        recipe definition RecGroup: arScrew[0].rRstmax : REAL; arScrew[0].rRstmin : REAL; arScrew[0].iCountCycle : INT; arScrew[0].iActuatorsMove : INT; arScrew[0].iActuatorsStep : INT; arScrew[0].iActuatorsStartPos[0] : INT; arScrew[0].iActuatorsStartPos[1] : INT; arScrew[0].support[0].bPosition : BOOL; arScrew[0].support[0].arLength[0] : INT; arScrew[0].support[0].arLength[1] : INT; arScrew[0].support[0].name : WSTRING(20); arScrew[0].support[1].bPosition : BOOL; arScrew[0].support[1].arLength[0] : INT; arScrew[0].support[1].arLength[1] : INT; arScrew[0].support[1].name : WSTRING(20); arScrew[0].bDirRotate : BOOL; arScrew[0].rOut_diam : REAL; arScrew[0].rInner_diam : REAL; arScrew[0].rTurn_step : REAL; arScrew[0].rWidth : REAL; arScrew[0].rAngle_knives : REAL; arScrew[0].rMidle_line : REAL; arScrew[0].rInstal_support : REAL; arScrew[0].rPosX0 : REAL; arScrew[0].rPosX1 : REAL; arScrew[0].rPosX2 : REAL; arScrew[0].equip.place : WSTRING(10); arScrew[0].equip.name : WSTRING(20); arScrew[0].name : WSTRING(20); arScrew[1].rRstmax : REAL; arScrew[1].rRstmin : REAL; arScrew[1].iCountCycle : INT; arScrew[1].iActuatorsMove : INT; arScrew[1].iActuatorsStep : INT; arScrew[1].iActuatorsStartPos[0] : INT; arScrew[1].iActuatorsStartPos[1] : INT; arScrew[1].support[0].bPosition : BOOL; arScrew[1].support[0].arLength[0] : INT; arScrew[1].support[0].arLength[1] : INT; arScrew[1].support[0].name : WSTRING(20); arScrew[1].support[1].bPosition : BOOL; arScrew[1].support[1].arLength[0] : INT; arScrew[1].support[1].arLength[1] : INT; arScrew[1].support[1].name : WSTRING(20); arScrew[1].bDirRotate : BOOL; arScrew[1].rOut_diam : REAL; arScrew[1].rInner_diam : REAL; arScrew[1].rTurn_step : REAL; arScrew[1].rWidth : REAL; arScrew[1].rAngle_knives : REAL; arScrew[1].rMidle_line : REAL; arScrew[1].rInstal_support : REAL; arScrew[1].rPosX0 : REAL; arScrew[1].rPosX1 : REAL; arScrew[1].rPosX2 : REAL; arScrew[1].equip.place : WSTRING(10); arScrew[1].equip.name : WSTRING(20); arScrew[1].name : WSTRING(20); arScrew[2].rRstmax : REAL; arScrew[2].rRstmin : REAL; arScrew[2].iCountCycle : INT; arScrew[2].iActuatorsMove : INT; arScrew[2].iActuatorsStep : INT; arScrew[2].iActuatorsStartPos[0] : INT; arScrew[2].iActuatorsStartPos[1] : INT; arScrew[2].support[0].bPosition : BOOL; arScrew[2].support[0].arLength[0] : INT; arScrew[2].support[0].arLength[1] : INT; arScrew[2].support[0].name : WSTRING(20); arScrew[2].support[1].bPosition : BOOL; arScrew[2].support[1].arLength[0] : INT; arScrew[2].support[1].arLength[1] : INT; arScrew[2].support[1].name : WSTRING(20); arScrew[2].bDirRotate : BOOL; arScrew[2].rOut_diam : REAL; arScrew[2].rInner_diam : REAL; arScrew[2].rTurn_step : REAL; arScrew[2].rWidth : REAL; arScrew[2].rAngle_knives : REAL; arScrew[2].rMidle_line : REAL; arScrew[2].rInstal_support : REAL; arScrew[2].rPosX0 : REAL; arScrew[2].rPosX1 : REAL; arScrew[2].rPosX2 : REAL; arScrew[2].equip.place : WSTRING(10); arScrew[2].equip.name : WSTRING(20); arScrew[2].name : WSTRING(20); arScrew[3].rRstmax : REAL; arScrew[3].rRstmin : REAL; arScrew[3].iCountCycle : INT; arScrew[3].iActuatorsMove : INT; arScrew[3].iActuatorsStep : INT; arScrew[3].iActuatorsStartPos[0] : INT; arScrew[3].iActuatorsStartPos[1] : INT; arScrew[3].support[0].bPosition : BOOL; arScrew[3].support[0].arLength[0] : INT; arScrew[3].support[0].arLength[1] : INT; arScrew[3].support[0].name : WSTRING(20); arScrew[3].support[1].bPosition : BOOL; arScrew[3].support[1].arLength[0] : INT; arScrew[3].support[1].arLength[1] : INT; arScrew[3].support[1].name : WSTRING(20); arScrew[3].bDirRotate : BOOL; arScrew[3].rOut_diam : REAL; arScrew[3].rInner_diam : REAL; arScrew[3].rTurn_step : REAL; arScrew[3].rWidth : REAL; arScrew[3].rAngle_knives : REAL; arScrew[3].rMidle_line : REAL; arScrew[3].rInstal_support : REAL; arScrew[3].rPosX0 : REAL; arScrew[3].rPosX1 : REAL; arScrew[3].rPosX2 : REAL; arScrew[3].equip.place : WSTRING(10); arScrew[3].equip.name : WSTRING(20); arScrew[3].name : WSTRING(20); arScrew[4].rRstmax : REAL; arScrew[4].rRstmin : REAL; arScrew[4].iCountCycle : INT; arScrew[4].iActuatorsMove : INT; arScrew[4].iActuatorsStep : INT; arScrew[4].iActuatorsStartPos[0] : INT; arScrew[4].iActuatorsStartPos[1] : INT; arScrew[4].support[0].bPosition : BOOL; arScrew[4].support[0].arLength[0] : INT; arScrew[4].support[0].arLength[1] : INT; arScrew[4].support[0].name : WSTRING(20); arScrew[4].support[1].bPosition : BOOL; arScrew[4].support[1].arLength[0] : INT; arScrew[4].support[1].arLength[1] : INT; arScrew[4].support[1].name : WSTRING(20); arScrew[4].bDirRotate : BOOL; arScrew[4].rOut_diam : REAL; arScrew[4].rInner_diam : REAL; arScrew[4].rTurn_step : REAL; arScrew[4].rWidth : REAL; arScrew[4].rAngle_knives : REAL; arScrew[4].rMidle_line : REAL; arScrew[4].rInstal_support : REAL; arScrew[4].rPosX0 : REAL; arScrew[4].rPosX1 : REAL; arScrew[4].rPosX2 : REAL; arScrew[4].equip.place : WSTRING(10); arScrew[4].equip.name : WSTRING(20); arScrew[4].name : WSTRING(20); arScrew[5].rRstmax : REAL; arScrew[5].rRstmin : REAL; arScrew[5].iCountCycle : INT; arScrew[5].iActuatorsMove : INT; arScrew[5].iActuatorsStep : INT; arScrew[5].iActuatorsStartPos[0] : INT; arScrew[5].iActuatorsStartPos[1] : INT; arScrew[5].support[0].bPosition : BOOL; arScrew[5].support[0].arLength[0] : INT; arScrew[5].support[0].arLength[1] : INT; arScrew[5].support[0].name : WSTRING(20); arScrew[5].support[1].bPosition : BOOL; arScrew[5].support[1].arLength[0] : INT; arScrew[5].support[1].arLength[1] : INT; arScrew[5].support[1].name : WSTRING(20); arScrew[5].bDirRotate : BOOL; arScrew[5].rOut_diam : REAL; arScrew[5].rInner_diam : REAL; arScrew[5].rTurn_step : REAL; arScrew[5].rWidth : REAL; arScrew[5].rAngle_knives : REAL; arScrew[5].rMidle_line : REAL; arScrew[5].rInstal_support : REAL; arScrew[5].rPosX0 : REAL; arScrew[5].rPosX1 : REAL; arScrew[5].rPosX2 : REAL; arScrew[5].equip.place : WSTRING(10); arScrew[5].equip.name : WSTRING(20); arScrew[5].name : WSTRING(20); arScrew[6].rRstmax : REAL; arScrew[6].rRstmin : REAL; arScrew[6].iCountCycle : INT; arScrew[6].iActuatorsMove : INT; arScrew[6].iActuatorsStep : INT; arScrew[6].iActuatorsStartPos[0] : INT; arScrew[6].iActuatorsStartPos[1] : INT; arScrew[6].support[0].bPosition : BOOL; arScrew[6].support[0].arLength[0] : INT; arScrew[6].support[0].arLength[1] : INT; arScrew[6].support[0].name : WSTRING(20); arScrew[6].support[1].bPosition : BOOL; arScrew[6].support[1].arLength[0] : INT; arScrew[6].support[1].arLength[1] : INT; arScrew[6].support[1].name : WSTRING(20); arScrew[6].bDirRotate : BOOL; arScrew[6].rOut_diam : REAL; arScrew[6].rInner_diam : REAL; arScrew[6].rTurn_step : REAL; arScrew[6].rWidth : REAL; arScrew[6].rAngle_knives : REAL; arScrew[6].rMidle_line : REAL; arScrew[6].rInstal_support : REAL; arScrew[6].rPosX0 : REAL; arScrew[6].rPosX1 : REAL; arScrew[6].rPosX2 : REAL; arScrew[6].equip.place : WSTRING(10); arScrew[6].equip.name : WSTRING(20); arScrew[6].name : WSTRING(20); arScrew[7].rRstmax : REAL; arScrew[7].rRstmin : REAL; arScrew[7].iCountCycle : INT; arScrew[7].iActuatorsMove : INT; arScrew[7].iActuatorsStep : INT; arScrew[7].iActuatorsStartPos[0] : INT; arScrew[7].iActuatorsStartPos[1] : INT; arScrew[7].support[0].bPosition : BOOL; arScrew[7].support[0].arLength[0] : INT; arScrew[7].support[0].arLength[1] : INT; arScrew[7].support[0].name : WSTRING(20); arScrew[7].support[1].bPosition : BOOL; arScrew[7].support[1].arLength[0] : INT; arScrew[7].support[1].arLength[1] : INT; arScrew[7].support[1].name : WSTRING(20); arScrew[7].bDirRotate : BOOL; arScrew[7].rOut_diam : REAL; arScrew[7].rInner_diam : REAL; arScrew[7].rTurn_step : REAL; arScrew[7].rWidth : REAL; arScrew[7].rAngle_knives : REAL; arScrew[7].rMidle_line : REAL; arScrew[7].rInstal_support : REAL; arScrew[7].rPosX0 : REAL; arScrew[7].rPosX1 : REAL; arScrew[7].rPosX2 : REAL; arScrew[7].equip.place : WSTRING(10); arScrew[7].equip.name : WSTRING(20); arScrew[7].name : WSTRING(20); arScrew[8].rRstmax : REAL; arScrew[8].rRstmin : REAL; arScrew[8].iCountCycle : INT; arScrew[8].iActuatorsMove : INT; arScrew[8].iActuatorsStep : INT; arScrew[8].iActuatorsStartPos[0] : INT; arScrew[8].iActuatorsStartPos[1] : INT; arScrew[8].support[0].bPosition : BOOL; arScrew[8].support[0].arLength[0] : INT; arScrew[8].support[0].arLength[1] : INT; arScrew[8].support[0].name : WSTRING(20); arScrew[8].support[1].bPosition : BOOL; arScrew[8].support[1].arLength[0] : INT; arScrew[8].support[1].arLength[1] : INT; arScrew[8].support[1].name : WSTRING(20); arScrew[8].bDirRotate : BOOL; arScrew[8].rOut_diam : REAL; arScrew[8].rInner_diam : REAL; arScrew[8].rTurn_step : REAL; arScrew[8].rWidth : REAL; arScrew[8].rAngle_knives : REAL; arScrew[8].rMidle_line : REAL; arScrew[8].rInstal_support : REAL; arScrew[8].rPosX0 : REAL; arScrew[8].rPosX1 : REAL; arScrew[8].rPosX2 : REAL; arScrew[8].equip.place : WSTRING(10); arScrew[8].equip.name : WSTRING(20); arScrew[8].name : WSTRING(20); arScrew[9].rRstmax : REAL; arScrew[9].rRstmin : REAL; arScrew[9].iCountCycle : INT; arScrew[9].iActuatorsMove : INT; arScrew[9].iActuatorsStep : INT; arScrew[9].iActuatorsStartPos[0] : INT; arScrew[9].iActuatorsStartPos[1] : INT; arScrew[9].support[0].bPosition : BOOL; arScrew[9].support[0].arLength[0] : INT; arScrew[9].support[0].arLength[1] : INT; arScrew[9].support[0].name : WSTRING(20); arScrew[9].support[1].bPosition : BOOL; arScrew[9].support[1].arLength[0] : INT; arScrew[9].support[1].arLength[1] : INT; arScrew[9].support[1].name : WSTRING(20); arScrew[9].bDirRotate : BOOL; arScrew[9].rOut_diam : REAL; arScrew[9].rInner_diam : REAL; arScrew[9].rTurn_step : REAL; arScrew[9].rWidth : REAL; arScrew[9].rAngle_knives : REAL; arScrew[9].rMidle_line : REAL; arScrew[9].rInstal_support : REAL; arScrew[9].rPosX0 : REAL; arScrew[9].rPosX1 : REAL; arScrew[9].rPosX2 : REAL; arScrew[9].equip.place : WSTRING(10); arScrew[9].equip.name : WSTRING(20); arScrew[9].name : WSTRING(20); arScrew[10].rRstmax : REAL; arScrew[10].rRstmin : REAL; arScrew[10].iCountCycle : INT; arScrew[10].iActuatorsMove : INT; arScrew[10].iActuatorsStep : INT; arScrew[10].iActuatorsStartPos[0] : INT; arScrew[10].iActuatorsStartPos[1] : INT; arScrew[10].support[0].bPosition : BOOL; arScrew[10].support[0].arLength[0] : INT; arScrew[10].support[0].arLength[1] : INT; arScrew[10].support[0].name : WSTRING(20); arScrew[10].support[1].bPosition : BOOL; arScrew[10].support[1].arLength[0] : INT; arScrew[10].support[1].arLength[1] : INT; arScrew[10].support[1].name : WSTRING(20); arScrew[10].bDirRotate : BOOL; arScrew[10].rOut_diam : REAL; arScrew[10].rInner_diam : REAL; arScrew[10].rTurn_step : REAL; arScrew[10].rWidth : REAL; arScrew[10].rAngle_knives : REAL; arScrew[10].rMidle_line : REAL; arScrew[10].rInstal_support : REAL; arScrew[10].rPosX0 : REAL; arScrew[10].rPosX1 : REAL; arScrew[10].rPosX2 : REAL; arScrew[10].equip.place : WSTRING(10); arScrew[10].equip.name : WSTRING(20); arScrew[10].name : WSTRING(20); arScrew[11].rRstmax : REAL; arScrew[11].rRstmin : REAL; arScrew[11].iCountCycle : INT; arScrew[11].iActuatorsMove : INT; arScrew[11].iActuatorsStep : INT; arScrew[11].iActuatorsStartPos[0] : INT; arScrew[11].iActuatorsStartPos[1] : INT; arScrew[11].support[0].bPosition : BOOL; arScrew[11].support[0].arLength[0] : INT; arScrew[11].support[0].arLength[1] : INT; arScrew[11].support[0].name : WSTRING(20); arScrew[11].support[1].bPosition : BOOL; arScrew[11].support[1].arLength[0] : INT; arScrew[11].support[1].arLength[1] : INT; arScrew[11].support[1].name : WSTRING(20); arScrew[11].bDirRotate : BOOL; arScrew[11].rOut_diam : REAL; arScrew[11].rInner_diam : REAL; arScrew[11].rTurn_step : REAL; arScrew[11].rWidth : REAL; arScrew[11].rAngle_knives : REAL; arScrew[11].rMidle_line : REAL; arScrew[11].rInstal_support : REAL; arScrew[11].rPosX0 : REAL; arScrew[11].rPosX1 : REAL; arScrew[11].rPosX2 : REAL; arScrew[11].equip.place : WSTRING(10); arScrew[11].equip.name : WSTRING(20); arScrew[11].name : WSTRING(20); arScrew[12].rRstmax : REAL; arScrew[12].rRstmin : REAL; arScrew[12].iCountCycle : INT; arScrew[12].iActuatorsMove : INT; arScrew[12].iActuatorsStep : INT; arScrew[12].iActuatorsStartPos[0] : INT; arScrew[12].iActuatorsStartPos[1] : INT; arScrew[12].support[0].bPosition : BOOL; arScrew[12].support[0].arLength[0] : INT; arScrew[12].support[0].arLength[1] : INT; arScrew[12].support[0].name : WSTRING(20); arScrew[12].support[1].bPosition : BOOL; arScrew[12].support[1].arLength[0] : INT; arScrew[12].support[1].arLength[1] : INT; arScrew[12].support[1].name : WSTRING(20); arScrew[12].bDirRotate : BOOL; arScrew[12].rOut_diam : REAL; arScrew[12].rInner_diam : REAL; arScrew[12].rTurn_step : REAL; arScrew[12].rWidth : REAL; arScrew[12].rAngle_knives : REAL; arScrew[12].rMidle_line : REAL; arScrew[12].rInstal_support : REAL; arScrew[12].rPosX0 : REAL; arScrew[12].rPosX1 : REAL; arScrew[12].rPosX2 : REAL; arScrew[12].equip.place : WSTRING(10); arScrew[12].equip.name : WSTRING(20); arScrew[12].name : WSTRING(20); arScrew[13].rRstmax : REAL; arScrew[13].rRstmin : REAL; arScrew[13].iCountCycle : INT; arScrew[13].iActuatorsMove : INT; arScrew[13].iActuatorsStep : INT; arScrew[13].iActuatorsStartPos[0] : INT; arScrew[13].iActuatorsStartPos[1] : INT; arScrew[13].support[0].bPosition : BOOL; arScrew[13].support[0].arLength[0] : INT; arScrew[13].support[0].arLength[1] : INT; arScrew[13].support[0].name : WSTRING(20); arScrew[13].support[1].bPosition : BOOL; arScrew[13].support[1].arLength[0] : INT; arScrew[13].support[1].arLength[1] : INT; arScrew[13].support[1].name : WSTRING(20); arScrew[13].bDirRotate : BOOL; arScrew[13].rOut_diam : REAL; arScrew[13].rInner_diam : REAL; arScrew[13].rTurn_step : REAL; arScrew[13].rWidth : REAL; arScrew[13].rAngle_knives : REAL; arScrew[13].rMidle_line : REAL; arScrew[13].rInstal_support : REAL; arScrew[13].rPosX0 : REAL; arScrew[13].rPosX1 : REAL; arScrew[13].rPosX2 : REAL; arScrew[13].equip.place : WSTRING(10); arScrew[13].equip.name : WSTRING(20); arScrew[13].name : WSTRING(20); arScrew[14].rRstmax : REAL; arScrew[14].rRstmin : REAL; arScrew[14].iCountCycle : INT; arScrew[14].iActuatorsMove : INT; arScrew[14].iActuatorsStep : INT; arScrew[14].iActuatorsStartPos[0] : INT; arScrew[14].iActuatorsStartPos[1] : INT; arScrew[14].support[0].bPosition : BOOL; arScrew[14].support[0].arLength[0] : INT; arScrew[14].support[0].arLength[1] : INT; arScrew[14].support[0].name : WSTRING(20); arScrew[14].support[1].bPosition : BOOL; arScrew[14].support[1].arLength[0] : INT; arScrew[14].support[1].arLength[1] : INT; arScrew[14].support[1].name : WSTRING(20); arScrew[14].bDirRotate : BOOL; arScrew[14].rOut_diam : REAL; arScrew[14].rInner_diam : REAL; arScrew[14].rTurn_step : REAL; arScrew[14].rWidth : REAL; arScrew[14].rAngle_knives : REAL; arScrew[14].rMidle_line : REAL; arScrew[14].rInstal_support : REAL; arScrew[14].rPosX0 : REAL; arScrew[14].rPosX1 : REAL; arScrew[14].rPosX2 : REAL; arScrew[14].equip.place : WSTRING(10); arScrew[14].equip.name : WSTRING(20); arScrew[14].name : WSTRING(20); arScrew[15].rRstmax : REAL; arScrew[15].rRstmin : REAL; arScrew[15].iCountCycle : INT; arScrew[15].iActuatorsMove : INT; arScrew[15].iActuatorsStep : INT; arScrew[15].iActuatorsStartPos[0] : INT; arScrew[15].iActuatorsStartPos[1] : INT; arScrew[15].support[0].bPosition : BOOL; arScrew[15].support[0].arLength[0] : INT; arScrew[15].support[0].arLength[1] : INT; arScrew[15].support[0].name : WSTRING(20); arScrew[15].support[1].bPosition : BOOL; arScrew[15].support[1].arLength[0] : INT; arScrew[15].support[1].arLength[1] : INT; arScrew[15].support[1].name : WSTRING(20); arScrew[15].bDirRotate : BOOL; arScrew[15].rOut_diam : REAL; arScrew[15].rInner_diam : REAL; arScrew[15].rTurn_step : REAL; arScrew[15].rWidth : REAL; arScrew[15].rAngle_knives : REAL; arScrew[15].rMidle_line : REAL; arScrew[15].rInstal_support : REAL; arScrew[15].rPosX0 : REAL; arScrew[15].rPosX1 : REAL; arScrew[15].rPosX2 : REAL; arScrew[15].equip.place : WSTRING(10); arScrew[15].equip.name : WSTRING(20); arScrew[15].name : WSTRING(20); arScrew[16].rRstmax : REAL; arScrew[16].rRstmin : REAL; arScrew[16].iCountCycle : INT; arScrew[16].iActuatorsMove : INT; arScrew[16].iActuatorsStep : INT; arScrew[16].iActuatorsStartPos[0] : INT; arScrew[16].iActuatorsStartPos[1] : INT; arScrew[16].support[0].bPosition : BOOL; arScrew[16].support[0].arLength[0] : INT; arScrew[16].support[0].arLength[1] : INT; arScrew[16].support[0].name : WSTRING(20); arScrew[16].support[1].bPosition : BOOL; arScrew[16].support[1].arLength[0] : INT; arScrew[16].support[1].arLength[1] : INT; arScrew[16].support[1].name : WSTRING(20); arScrew[16].bDirRotate : BOOL; arScrew[16].rOut_diam : REAL; arScrew[16].rInner_diam : REAL; arScrew[16].rTurn_step : REAL; arScrew[16].rWidth : REAL; arScrew[16].rAngle_knives : REAL; arScrew[16].rMidle_line : REAL; arScrew[16].rInstal_support : REAL; arScrew[16].rPosX0 : REAL; arScrew[16].rPosX1 : REAL; arScrew[16].rPosX2 : REAL; arScrew[16].equip.place : WSTRING(10); arScrew[16].equip.name : WSTRING(20); arScrew[16].name : WSTRING(20); arScrew[17].rRstmax : REAL; arScrew[17].rRstmin : REAL; arScrew[17].iCountCycle : INT; arScrew[17].iActuatorsMove : INT; arScrew[17].iActuatorsStep : INT; arScrew[17].iActuatorsStartPos[0] : INT; arScrew[17].iActuatorsStartPos[1] : INT; arScrew[17].support[0].bPosition : BOOL; arScrew[17].support[0].arLength[0] : INT; arScrew[17].support[0].arLength[1] : INT; arScrew[17].support[0].name : WSTRING(20); arScrew[17].support[1].bPosition : BOOL; arScrew[17].support[1].arLength[0] : INT; arScrew[17].support[1].arLength[1] : INT; arScrew[17].support[1].name : WSTRING(20); arScrew[17].bDirRotate : BOOL; arScrew[17].rOut_diam : REAL; arScrew[17].rInner_diam : REAL; arScrew[17].rTurn_step : REAL; arScrew[17].rWidth : REAL; arScrew[17].rAngle_knives : REAL; arScrew[17].rMidle_line : REAL; arScrew[17].rInstal_support : REAL; arScrew[17].rPosX0 : REAL; arScrew[17].rPosX1 : REAL; arScrew[17].rPosX2 : REAL; arScrew[17].equip.place : WSTRING(10); arScrew[17].equip.name : WSTRING(20); arScrew[17].name : WSTRING(20); arScrew[18].rRstmax : REAL; arScrew[18].rRstmin : REAL; arScrew[18].iCountCycle : INT; arScrew[18].iActuatorsMove : INT; arScrew[18].iActuatorsStep : INT; arScrew[18].iActuatorsStartPos[0] : INT; arScrew[18].iActuatorsStartPos[1] : INT; arScrew[18].support[0].bPosition : BOOL; arScrew[18].support[0].arLength[0] : INT; arScrew[18].support[0].arLength[1] : INT; arScrew[18].support[0].name : WSTRING(20); arScrew[18].support[1].bPosition : BOOL; arScrew[18].support[1].arLength[0] : INT; arScrew[18].support[1].arLength[1] : INT; arScrew[18].support[1].name : WSTRING(20); arScrew[18].bDirRotate : BOOL; arScrew[18].rOut_diam : REAL; arScrew[18].rInner_diam : REAL; arScrew[18].rTurn_step : REAL; arScrew[18].rWidth : REAL; arScrew[18].rAngle_knives : REAL; arScrew[18].rMidle_line : REAL; arScrew[18].rInstal_support : REAL; arScrew[18].rPosX0 : REAL; arScrew[18].rPosX1 : REAL; arScrew[18].rPosX2 : REAL; arScrew[18].equip.place : WSTRING(10); arScrew[18].equip.name : WSTRING(20); arScrew[18].name : WSTRING(20); arScrew[19].rRstmax : REAL; arScrew[19].rRstmin : REAL; arScrew[19].iCountCycle : INT; arScrew[19].iActuatorsMove : INT; arScrew[19].iActuatorsStep : INT; arScrew[19].iActuatorsStartPos[0] : INT; arScrew[19].iActuatorsStartPos[1] : INT; arScrew[19].support[0].bPosition : BOOL; arScrew[19].support[0].arLength[0] : INT; arScrew[19].support[0].arLength[1] : INT; arScrew[19].support[0].name : WSTRING(20); arScrew[19].support[1].bPosition : BOOL; arScrew[19].support[1].arLength[0] : INT; arScrew[19].support[1].arLength[1] : INT; arScrew[19].support[1].name : WSTRING(20); arScrew[19].bDirRotate : BOOL; arScrew[19].rOut_diam : REAL; arScrew[19].rInner_diam : REAL; arScrew[19].rTurn_step : REAL; arScrew[19].rWidth : REAL; arScrew[19].rAngle_knives : REAL; arScrew[19].rMidle_line : REAL; arScrew[19].rInstal_support : REAL; arScrew[19].rPosX0 : REAL; arScrew[19].rPosX1 : REAL; arScrew[19].rPosX2 : REAL; arScrew[19].equip.place : WSTRING(10); arScrew[19].equip.name : WSTRING(20); arScrew[19].name : WSTRING(20); arScrew[20].rRstmax : REAL; arScrew[20].rRstmin : REAL; arScrew[20].iCountCycle : INT; arScrew[20].iActuatorsMove : INT; arScrew[20].iActuatorsStep : INT; arScrew[20].iActuatorsStartPos[0] : INT; arScrew[20].iActuatorsStartPos[1] : INT; arScrew[20].support[0].bPosition : BOOL; arScrew[20].support[0].arLength[0] : INT; arScrew[20].support[0].arLength[1] : INT; arScrew[20].support[0].name : WSTRING(20); arScrew[20].support[1].bPosition : BOOL; arScrew[20].support[1].arLength[0] : INT; arScrew[20].support[1].arLength[1] : INT; arScrew[20].support[1].name : WSTRING(20); arScrew[20].bDirRotate : BOOL; arScrew[20].rOut_diam : REAL; arScrew[20].rInner_diam : REAL; arScrew[20].rTurn_step : REAL; arScrew[20].rWidth : REAL; arScrew[20].rAngle_knives : REAL; arScrew[20].rMidle_line : REAL; arScrew[20].rInstal_support : REAL; arScrew[20].rPosX0 : REAL; arScrew[20].rPosX1 : REAL; arScrew[20].rPosX2 : REAL; arScrew[20].equip.place : WSTRING(10); arScrew[20].equip.name : WSTRING(20); arScrew[20].name : WSTRING(20); arScrew[21].rRstmax : REAL; arScrew[21].rRstmin : REAL; arScrew[21].iCountCycle : INT; arScrew[21].iActuatorsMove : INT; arScrew[21].iActuatorsStep : INT; arScrew[21].iActuatorsStartPos[0] : INT; arScrew[21].iActuatorsStartPos[1] : INT; arScrew[21].support[0].bPosition : BOOL; arScrew[21].support[0].arLength[0] : INT; arScrew[21].support[0].arLength[1] : INT; arScrew[21].support[0].name : WSTRING(20); arScrew[21].support[1].bPosition : BOOL; arScrew[21].support[1].arLength[0] : INT; arScrew[21].support[1].arLength[1] : INT; arScrew[21].support[1].name : WSTRING(20); arScrew[21].bDirRotate : BOOL; arScrew[21].rOut_diam : REAL; arScrew[21].rInner_diam : REAL; arScrew[21].rTurn_step : REAL; arScrew[21].rWidth : REAL; arScrew[21].rAngle_knives : REAL; arScrew[21].rMidle_line : REAL; arScrew[21].rInstal_support : REAL; arScrew[21].rPosX0 : REAL; arScrew[21].rPosX1 : REAL; arScrew[21].rPosX2 : REAL; arScrew[21].equip.place : WSTRING(10); arScrew[21].equip.name : WSTRING(20); arScrew[21].name : WSTRING(20); arScrew[22].rRstmax : REAL; arScrew[22].rRstmin : REAL; arScrew[22].iCountCycle : INT; arScrew[22].iActuatorsMove : INT; arScrew[22].iActuatorsStep : INT; arScrew[22].iActuatorsStartPos[0] : INT; arScrew[22].iActuatorsStartPos[1] : INT; arScrew[22].support[0].bPosition : BOOL; arScrew[22].support[0].arLength[0] : INT; arScrew[22].support[0].arLength[1] : INT; arScrew[22].support[0].name : WSTRING(20); arScrew[22].support[1].bPosition : BOOL; arScrew[22].support[1].arLength[0] : INT; arScrew[22].support[1].arLength[1] : INT; arScrew[22].support[1].name : WSTRING(20); arScrew[22].bDirRotate : BOOL; arScrew[22].rOut_diam : REAL; arScrew[22].rInner_diam : REAL; arScrew[22].rTurn_step : REAL; arScrew[22].rWidth : REAL; arScrew[22].rAngle_knives : REAL; arScrew[22].rMidle_line : REAL; arScrew[22].rInstal_support : REAL; arScrew[22].rPosX0 : REAL; arScrew[22].rPosX1 : REAL; arScrew[22].rPosX2 : REAL; arScrew[22].equip.place : WSTRING(10); arScrew[22].equip.name : WSTRING(20); arScrew[22].name : WSTRING(20); arScrew[23].rRstmax : REAL; arScrew[23].rRstmin : REAL; arScrew[23].iCountCycle : INT; arScrew[23].iActuatorsMove : INT; arScrew[23].iActuatorsStep : INT; arScrew[23].iActuatorsStartPos[0] : INT; arScrew[23].iActuatorsStartPos[1] : INT; arScrew[23].support[0].bPosition : BOOL; arScrew[23].support[0].arLength[0] : INT; arScrew[23].support[0].arLength[1] : INT; arScrew[23].support[0].name : WSTRING(20); arScrew[23].support[1].bPosition : BOOL; arScrew[23].support[1].arLength[0] : INT; arScrew[23].support[1].arLength[1] : INT; arScrew[23].support[1].name : WSTRING(20); arScrew[23].bDirRotate : BOOL; arScrew[23].rOut_diam : REAL; arScrew[23].rInner_diam : REAL; arScrew[23].rTurn_step : REAL; arScrew[23].rWidth : REAL; arScrew[23].rAngle_knives : REAL; arScrew[23].rMidle_line : REAL; arScrew[23].rInstal_support : REAL; arScrew[23].rPosX0 : REAL; arScrew[23].rPosX1 : REAL; arScrew[23].rPosX2 : REAL; arScrew[23].equip.place : WSTRING(10); arScrew[23].equip.name : WSTRING(20); arScrew[23].name : WSTRING(20); arScrew[24].rRstmax : REAL; arScrew[24].rRstmin : REAL; arScrew[24].iCountCycle : INT; arScrew[24].iActuatorsMove : INT; arScrew[24].iActuatorsStep : INT; arScrew[24].iActuatorsStartPos[0] : INT; arScrew[24].iActuatorsStartPos[1] : INT; arScrew[24].support[0].bPosition : BOOL; arScrew[24].support[0].arLength[0] : INT; arScrew[24].support[0].arLength[1] : INT; arScrew[24].support[0].name : WSTRING(20); arScrew[24].support[1].bPosition : BOOL; arScrew[24].support[1].arLength[0] : INT; arScrew[24].support[1].arLength[1] : INT; arScrew[24].support[1].name : WSTRING(20); arScrew[24].bDirRotate : BOOL; arScrew[24].rOut_diam : REAL; arScrew[24].rInner_diam : REAL; arScrew[24].rTurn_step : REAL; arScrew[24].rWidth : REAL; arScrew[24].rAngle_knives : REAL; arScrew[24].rMidle_line : REAL; arScrew[24].rInstal_support : REAL; arScrew[24].rPosX0 : REAL; arScrew[24].rPosX1 : REAL; arScrew[24].rPosX2 : REAL; arScrew[24].equip.place : WSTRING(10); arScrew[24].equip.name : WSTRING(20); arScrew[24].name : WSTRING(20); arScrew[25].rRstmax : REAL; arScrew[25].rRstmin : REAL; arScrew[25].iCountCycle : INT; arScrew[25].iActuatorsMove : INT; arScrew[25].iActuatorsStep : INT; arScrew[25].iActuatorsStartPos[0] : INT; arScrew[25].iActuatorsStartPos[1] : INT; arScrew[25].support[0].bPosition : BOOL; arScrew[25].support[0].arLength[0] : INT; arScrew[25].support[0].arLength[1] : INT; arScrew[25].support[0].name : WSTRING(20); arScrew[25].support[1].bPosition : BOOL; arScrew[25].support[1].arLength[0] : INT; arScrew[25].support[1].arLength[1] : INT; arScrew[25].support[1].name : WSTRING(20); arScrew[25].bDirRotate : BOOL; arScrew[25].rOut_diam : REAL; arScrew[25].rInner_diam : REAL; arScrew[25].rTurn_step : REAL; arScrew[25].rWidth : REAL; arScrew[25].rAngle_knives : REAL; arScrew[25].rMidle_line : REAL; arScrew[25].rInstal_support : REAL; arScrew[25].rPosX0 : REAL; arScrew[25].rPosX1 : REAL; arScrew[25].rPosX2 : REAL; arScrew[25].equip.place : WSTRING(10); arScrew[25].equip.name : WSTRING(20); arScrew[25].name : WSTRING(20); arScrew[26].rRstmax : REAL; arScrew[26].rRstmin : REAL; arScrew[26].iCountCycle : INT; arScrew[26].iActuatorsMove : INT; arScrew[26].iActuatorsStep : INT; arScrew[26].iActuatorsStartPos[0] : INT; arScrew[26].iActuatorsStartPos[1] : INT; arScrew[26].support[0].bPosition : BOOL; arScrew[26].support[0].arLength[0] : INT; arScrew[26].support[0].arLength[1] : INT; arScrew[26].support[0].name : WSTRING(20); arScrew[26].support[1].bPosition : BOOL; arScrew[26].support[1].arLength[0] : INT; arScrew[26].support[1].arLength[1] : INT; arScrew[26].support[1].name : WSTRING(20); arScrew[26].bDirRotate : BOOL; arScrew[26].rOut_diam : REAL; arScrew[26].rInner_diam : REAL; arScrew[26].rTurn_step : REAL; arScrew[26].rWidth : REAL; arScrew[26].rAngle_knives : REAL; arScrew[26].rMidle_line : REAL; arScrew[26].rInstal_support : REAL; arScrew[26].rPosX0 : REAL; arScrew[26].rPosX1 : REAL; arScrew[26].rPosX2 : REAL; arScrew[26].equip.place : WSTRING(10); arScrew[26].equip.name : WSTRING(20); arScrew[26].name : WSTRING(20); arScrew[27].rRstmax : REAL; arScrew[27].rRstmin : REAL; arScrew[27].iCountCycle : INT; arScrew[27].iActuatorsMove : INT; arScrew[27].iActuatorsStep : INT; arScrew[27].iActuatorsStartPos[0] : INT; arScrew[27].iActuatorsStartPos[1] : INT; arScrew[27].support[0].bPosition : BOOL; arScrew[27].support[0].arLength[0] : INT; arScrew[27].support[0].arLength[1] : INT; arScrew[27].support[0].name : WSTRING(20); arScrew[27].support[1].bPosition : BOOL; arScrew[27].support[1].arLength[0] : INT; arScrew[27].support[1].arLength[1] : INT; arScrew[27].support[1].name : WSTRING(20); arScrew[27].bDirRotate : BOOL; arScrew[27].rOut_diam : REAL; arScrew[27].rInner_diam : REAL; arScrew[27].rTurn_step : REAL; arScrew[27].rWidth : REAL; arScrew[27].rAngle_knives : REAL; arScrew[27].rMidle_line : REAL; arScrew[27].rInstal_support : REAL; arScrew[27].rPosX0 : REAL; arScrew[27].rPosX1 : REAL; arScrew[27].rPosX2 : REAL; arScrew[27].equip.place : WSTRING(10); arScrew[27].equip.name : WSTRING(20); arScrew[27].name : WSTRING(20); arScrew[28].rRstmax : REAL; arScrew[28].rRstmin : REAL; arScrew[28].iCountCycle : INT; arScrew[28].iActuatorsMove : INT; arScrew[28].iActuatorsStep : INT; arScrew[28].iActuatorsStartPos[0] : INT; arScrew[28].iActuatorsStartPos[1] : INT; arScrew[28].support[0].bPosition : BOOL; arScrew[28].support[0].arLength[0] : INT; arScrew[28].support[0].arLength[1] : INT; arScrew[28].support[0].name : WSTRING(20); arScrew[28].support[1].bPosition : BOOL; arScrew[28].support[1].arLength[0] : INT; arScrew[28].support[1].arLength[1] : INT; arScrew[28].support[1].name : WSTRING(20); arScrew[28].bDirRotate : BOOL; arScrew[28].rOut_diam : REAL; arScrew[28].rInner_diam : REAL; arScrew[28].rTurn_step : REAL; arScrew[28].rWidth : REAL; arScrew[28].rAngle_knives : REAL; arScrew[28].rMidle_line : REAL; arScrew[28].rInstal_support : REAL; arScrew[28].rPosX0 : REAL; arScrew[28].rPosX1 : REAL; arScrew[28].rPosX2 : REAL; arScrew[28].equip.place : WSTRING(10); arScrew[28].equip.name : WSTRING(20); arScrew[28].name : WSTRING(20); arScrew[29].rRstmax : REAL; arScrew[29].rRstmin : REAL; arScrew[29].iCountCycle : INT; arScrew[29].iActuatorsMove : INT; arScrew[29].iActuatorsStep : INT; arScrew[29].iActuatorsStartPos[0] : INT; arScrew[29].iActuatorsStartPos[1] : INT; arScrew[29].support[0].bPosition : BOOL; arScrew[29].support[0].arLength[0] : INT; arScrew[29].support[0].arLength[1] : INT; arScrew[29].support[0].name : WSTRING(20); arScrew[29].support[1].bPosition : BOOL; arScrew[29].support[1].arLength[0] : INT; arScrew[29].support[1].arLength[1] : INT; arScrew[29].support[1].name : WSTRING(20); arScrew[29].bDirRotate : BOOL; arScrew[29].rOut_diam : REAL; arScrew[29].rInner_diam : REAL; arScrew[29].rTurn_step : REAL; arScrew[29].rWidth : REAL; arScrew[29].rAngle_knives : REAL; arScrew[29].rMidle_line : REAL; arScrew[29].rInstal_support : REAL; arScrew[29].rPosX0 : REAL; arScrew[29].rPosX1 : REAL; arScrew[29].rPosX2 : REAL; arScrew[29].equip.place : WSTRING(10); arScrew[29].equip.name : WSTRING(20); arScrew[29].name : WSTRING(20); arScrew[30].rRstmax : REAL; arScrew[30].rRstmin : REAL; arScrew[30].iCountCycle : INT; arScrew[30].iActuatorsMove : INT; arScrew[30].iActuatorsStep : INT; arScrew[30].iActuatorsStartPos[0] : INT; arScrew[30].iActuatorsStartPos[1] : INT; arScrew[30].support[0].bPosition : BOOL; arScrew[30].support[0].arLength[0] : INT; arScrew[30].support[0].arLength[1] : INT; arScrew[30].support[0].name : WSTRING(20); arScrew[30].support[1].bPosition : BOOL; arScrew[30].support[1].arLength[0] : INT; arScrew[30].support[1].arLength[1] : INT; arScrew[30].support[1].name : WSTRING(20); arScrew[30].bDirRotate : BOOL; arScrew[30].rOut_diam : REAL; arScrew[30].rInner_diam : REAL; arScrew[30].rTurn_step : REAL; arScrew[30].rWidth : REAL; arScrew[30].rAngle_knives : REAL; arScrew[30].rMidle_line : REAL; arScrew[30].rInstal_support : REAL; arScrew[30].rPosX0 : REAL; arScrew[30].rPosX1 : REAL; arScrew[30].rPosX2 : REAL; arScrew[30].equip.place : WSTRING(10); arScrew[30].equip.name : WSTRING(20); arScrew[30].name : WSTRING(20); arScrew[31].rRstmax : REAL; arScrew[31].rRstmin : REAL; arScrew[31].iCountCycle : INT; arScrew[31].iActuatorsMove : INT; arScrew[31].iActuatorsStep : INT; arScrew[31].iActuatorsStartPos[0] : INT; arScrew[31].iActuatorsStartPos[1] : INT; arScrew[31].support[0].bPosition : BOOL; arScrew[31].support[0].arLength[0] : INT; arScrew[31].support[0].arLength[1] : INT; arScrew[31].support[0].name : WSTRING(20); arScrew[31].support[1].bPosition : BOOL; arScrew[31].support[1].arLength[0] : INT; arScrew[31].support[1].arLength[1] : INT; arScrew[31].support[1].name : WSTRING(20); arScrew[31].bDirRotate : BOOL; arScrew[31].rOut_diam : REAL; arScrew[31].rInner_diam : REAL; arScrew[31].rTurn_step : REAL; arScrew[31].rWidth : REAL; arScrew[31].rAngle_knives : REAL; arScrew[31].rMidle_line : REAL; arScrew[31].rInstal_support : REAL; arScrew[31].rPosX0 : REAL; arScrew[31].rPosX1 : REAL; arScrew[31].rPosX2 : REAL; arScrew[31].equip.place : WSTRING(10); arScrew[31].equip.name : WSTRING(20); arScrew[31].name : WSTRING(20); arScrew[32].rRstmax : REAL; arScrew[32].rRstmin : REAL; arScrew[32].iCountCycle : INT; arScrew[32].iActuatorsMove : INT; arScrew[32].iActuatorsStep : INT; arScrew[32].iActuatorsStartPos[0] : INT; arScrew[32].iActuatorsStartPos[1] : INT; arScrew[32].support[0].bPosition : BOOL; arScrew[32].support[0].arLength[0] : INT; arScrew[32].support[0].arLength[1] : INT; arScrew[32].support[0].name : WSTRING(20); arScrew[32].support[1].bPosition : BOOL; arScrew[32].support[1].arLength[0] : INT; arScrew[32].support[1].arLength[1] : INT; arScrew[32].support[1].name : WSTRING(20); arScrew[32].bDirRotate : BOOL; arScrew[32].rOut_diam : REAL; arScrew[32].rInner_diam : REAL; arScrew[32].rTurn_step : REAL; arScrew[32].rWidth : REAL; arScrew[32].rAngle_knives : REAL; arScrew[32].rMidle_line : REAL; arScrew[32].rInstal_support : REAL; arScrew[32].rPosX0 : REAL; arScrew[32].rPosX1 : REAL; arScrew[32].rPosX2 : REAL; arScrew[32].equip.place : WSTRING(10); arScrew[32].equip.name : WSTRING(20); arScrew[32].name : WSTRING(20); arScrew[33].rRstmax : REAL; arScrew[33].rRstmin : REAL; arScrew[33].iCountCycle : INT; arScrew[33].iActuatorsMove : INT; arScrew[33].iActuatorsStep : INT; arScrew[33].iActuatorsStartPos[0] : INT; arScrew[33].iActuatorsStartPos[1] : INT; arScrew[33].support[0].bPosition : BOOL; arScrew[33].support[0].arLength[0] : INT; arScrew[33].support[0].arLength[1] : INT; arScrew[33].support[0].name : WSTRING(20); arScrew[33].support[1].bPosition : BOOL; arScrew[33].support[1].arLength[0] : INT; arScrew[33].support[1].arLength[1] : INT; arScrew[33].support[1].name : WSTRING(20); arScrew[33].bDirRotate : BOOL; arScrew[33].rOut_diam : REAL; arScrew[33].rInner_diam : REAL; arScrew[33].rTurn_step : REAL; arScrew[33].rWidth : REAL; arScrew[33].rAngle_knives : REAL; arScrew[33].rMidle_line : REAL; arScrew[33].rInstal_support : REAL; arScrew[33].rPosX0 : REAL; arScrew[33].rPosX1 : REAL; arScrew[33].rPosX2 : REAL; arScrew[33].equip.place : WSTRING(10); arScrew[33].equip.name : WSTRING(20); arScrew[33].name : WSTRING(20); arScrew[34].rRstmax : REAL; arScrew[34].rRstmin : REAL; arScrew[34].iCountCycle : INT; arScrew[34].iActuatorsMove : INT; arScrew[34].iActuatorsStep : INT; arScrew[34].iActuatorsStartPos[0] : INT; arScrew[34].iActuatorsStartPos[1] : INT; arScrew[34].support[0].bPosition : BOOL; arScrew[34].support[0].arLength[0] : INT; arScrew[34].support[0].arLength[1] : INT; arScrew[34].support[0].name : WSTRING(20); arScrew[34].support[1].bPosition : BOOL; arScrew[34].support[1].arLength[0] : INT; arScrew[34].support[1].arLength[1] : INT; arScrew[34].support[1].name : WSTRING(20); arScrew[34].bDirRotate : BOOL; arScrew[34].rOut_diam : REAL; arScrew[34].rInner_diam : REAL; arScrew[34].rTurn_step : REAL; arScrew[34].rWidth : REAL; arScrew[34].rAngle_knives : REAL; arScrew[34].rMidle_line : REAL; arScrew[34].rInstal_support : REAL; arScrew[34].rPosX0 : REAL; arScrew[34].rPosX1 : REAL; arScrew[34].rPosX2 : REAL; arScrew[34].equip.place : WSTRING(10); arScrew[34].equip.name : WSTRING(20); arScrew[34].name : WSTRING(20); arScrew[35].rRstmax : REAL; arScrew[35].rRstmin : REAL; arScrew[35].iCountCycle : INT; arScrew[35].iActuatorsMove : INT; arScrew[35].iActuatorsStep : INT; arScrew[35].iActuatorsStartPos[0] : INT; arScrew[35].iActuatorsStartPos[1] : INT; arScrew[35].support[0].bPosition : BOOL; arScrew[35].support[0].arLength[0] : INT; arScrew[35].support[0].arLength[1] : INT; arScrew[35].support[0].name : WSTRING(20); arScrew[35].support[1].bPosition : BOOL; arScrew[35].support[1].arLength[0] : INT; arScrew[35].support[1].arLength[1] : INT; arScrew[35].support[1].name : WSTRING(20); arScrew[35].bDirRotate : BOOL; arScrew[35].rOut_diam : REAL; arScrew[35].rInner_diam : REAL; arScrew[35].rTurn_step : REAL; arScrew[35].rWidth : REAL; arScrew[35].rAngle_knives : REAL; arScrew[35].rMidle_line : REAL; arScrew[35].rInstal_support : REAL; arScrew[35].rPosX0 : REAL; arScrew[35].rPosX1 : REAL; arScrew[35].rPosX2 : REAL; arScrew[35].equip.place : WSTRING(10); arScrew[35].equip.name : WSTRING(20); arScrew[35].name : WSTRING(20); arScrew[36].rRstmax : REAL; arScrew[36].rRstmin : REAL; arScrew[36].iCountCycle : INT; arScrew[36].iActuatorsMove : INT; arScrew[36].iActuatorsStep : INT; arScrew[36].iActuatorsStartPos[0] : INT; arScrew[36].iActuatorsStartPos[1] : INT; arScrew[36].support[0].bPosition : BOOL; arScrew[36].support[0].arLength[0] : INT; arScrew[36].support[0].arLength[1] : INT; arScrew[36].support[0].name : WSTRING(20); arScrew[36].support[1].bPosition : BOOL; arScrew[36].support[1].arLength[0] : INT; arScrew[36].support[1].arLength[1] : INT; arScrew[36].support[1].name : WSTRING(20); arScrew[36].bDirRotate : BOOL; arScrew[36].rOut_diam : REAL; arScrew[36].rInner_diam : REAL; arScrew[36].rTurn_step : REAL; arScrew[36].rWidth : REAL; arScrew[36].rAngle_knives : REAL; arScrew[36].rMidle_line : REAL; arScrew[36].rInstal_support : REAL; arScrew[36].rPosX0 : REAL; arScrew[36].rPosX1 : REAL; arScrew[36].rPosX2 : REAL; arScrew[36].equip.place : WSTRING(10); arScrew[36].equip.name : WSTRING(20); arScrew[36].name : WSTRING(20); arScrew[37].rRstmax : REAL; arScrew[37].rRstmin : REAL; arScrew[37].iCountCycle : INT; arScrew[37].iActuatorsMove : INT; arScrew[37].iActuatorsStep : INT; arScrew[37].iActuatorsStartPos[0] : INT; arScrew[37].iActuatorsStartPos[1] : INT; arScrew[37].support[0].bPosition : BOOL; arScrew[37].support[0].arLength[0] : INT; arScrew[37].support[0].arLength[1] : INT; arScrew[37].support[0].name : WSTRING(20); arScrew[37].support[1].bPosition : BOOL; arScrew[37].support[1].arLength[0] : INT; arScrew[37].support[1].arLength[1] : INT; arScrew[37].support[1].name : WSTRING(20); arScrew[37].bDirRotate : BOOL; arScrew[37].rOut_diam : REAL; arScrew[37].rInner_diam : REAL; arScrew[37].rTurn_step : REAL; arScrew[37].rWidth : REAL; arScrew[37].rAngle_knives : REAL; arScrew[37].rMidle_line : REAL; arScrew[37].rInstal_support : REAL; arScrew[37].rPosX0 : REAL; arScrew[37].rPosX1 : REAL; arScrew[37].rPosX2 : REAL; arScrew[37].equip.place : WSTRING(10); arScrew[37].equip.name : WSTRING(20); arScrew[37].name : WSTRING(20); arScrew[38].rRstmax : REAL; arScrew[38].rRstmin : REAL; arScrew[38].iCountCycle : INT; arScrew[38].iActuatorsMove : INT; arScrew[38].iActuatorsStep : INT; arScrew[38].iActuatorsStartPos[0] : INT; arScrew[38].iActuatorsStartPos[1] : INT; arScrew[38].support[0].bPosition : BOOL; arScrew[38].support[0].arLength[0] : INT; arScrew[38].support[0].arLength[1] : INT; arScrew[38].support[0].name : WSTRING(20); arScrew[38].support[1].bPosition : BOOL; arScrew[38].support[1].arLength[0] : INT; arScrew[38].support[1].arLength[1] : INT; arScrew[38].support[1].name : WSTRING(20); arScrew[38].bDirRotate : BOOL; arScrew[38].rOut_diam : REAL; arScrew[38].rInner_diam : REAL; arScrew[38].rTurn_step : REAL; arScrew[38].rWidth : REAL; arScrew[38].rAngle_knives : REAL; arScrew[38].rMidle_line : REAL; arScrew[38].rInstal_support : REAL; arScrew[38].rPosX0 : REAL; arScrew[38].rPosX1 : REAL; arScrew[38].rPosX2 : REAL; arScrew[38].equip.place : WSTRING(10); arScrew[38].equip.name : WSTRING(20); arScrew[38].name : WSTRING(20); arScrew[39].rRstmax : REAL; arScrew[39].rRstmin : REAL; arScrew[39].iCountCycle : INT; arScrew[39].iActuatorsMove : INT; arScrew[39].iActuatorsStep : INT; arScrew[39].iActuatorsStartPos[0] : INT; arScrew[39].iActuatorsStartPos[1] : INT; arScrew[39].support[0].bPosition : BOOL; arScrew[39].support[0].arLength[0] : INT; arScrew[39].support[0].arLength[1] : INT; arScrew[39].support[0].name : WSTRING(20); arScrew[39].support[1].bPosition : BOOL; arScrew[39].support[1].arLength[0] : INT; arScrew[39].support[1].arLength[1] : INT; arScrew[39].support[1].name : WSTRING(20); arScrew[39].bDirRotate : BOOL; arScrew[39].rOut_diam : REAL; arScrew[39].rInner_diam : REAL; arScrew[39].rTurn_step : REAL; arScrew[39].rWidth : REAL; arScrew[39].rAngle_knives : REAL; arScrew[39].rMidle_line : REAL; arScrew[39].rInstal_support : REAL; arScrew[39].rPosX0 : REAL; arScrew[39].rPosX1 : REAL; arScrew[39].rPosX2 : REAL; arScrew[39].equip.place : WSTRING(10); arScrew[39].equip.name : WSTRING(20); arScrew[39].name : WSTRING(20); arScrew[40].rRstmax : REAL; arScrew[40].rRstmin : REAL; arScrew[40].iCountCycle : INT; arScrew[40].iActuatorsMove : INT; arScrew[40].iActuatorsStep : INT; arScrew[40].iActuatorsStartPos[0] : INT; arScrew[40].iActuatorsStartPos[1] : INT; arScrew[40].support[0].bPosition : BOOL; arScrew[40].support[0].arLength[0] : INT; arScrew[40].support[0].arLength[1] : INT; arScrew[40].support[0].name : WSTRING(20); arScrew[40].support[1].bPosition : BOOL; arScrew[40].support[1].arLength[0] : INT; arScrew[40].support[1].arLength[1] : INT; arScrew[40].support[1].name : WSTRING(20); arScrew[40].bDirRotate : BOOL; arScrew[40].rOut_diam : REAL; arScrew[40].rInner_diam : REAL; arScrew[40].rTurn_step : REAL; arScrew[40].rWidth : REAL; arScrew[40].rAngle_knives : REAL; arScrew[40].rMidle_line : REAL; arScrew[40].rInstal_support : REAL; arScrew[40].rPosX0 : REAL; arScrew[40].rPosX1 : REAL; arScrew[40].rPosX2 : REAL; arScrew[40].equip.place : WSTRING(10); arScrew[40].equip.name : WSTRING(20); arScrew[40].name : WSTRING(20); arScrew[41].rRstmax : REAL; arScrew[41].rRstmin : REAL; arScrew[41].iCountCycle : INT; arScrew[41].iActuatorsMove : INT; arScrew[41].iActuatorsStep : INT; arScrew[41].iActuatorsStartPos[0] : INT; arScrew[41].iActuatorsStartPos[1] : INT; arScrew[41].support[0].bPosition : BOOL; arScrew[41].support[0].arLength[0] : INT; arScrew[41].support[0].arLength[1] : INT; arScrew[41].support[0].name : WSTRING(20); arScrew[41].support[1].bPosition : BOOL; arScrew[41].support[1].arLength[0] : INT; arScrew[41].support[1].arLength[1] : INT; arScrew[41].support[1].name : WSTRING(20); arScrew[41].bDirRotate : BOOL; arScrew[41].rOut_diam : REAL; arScrew[41].rInner_diam : REAL; arScrew[41].rTurn_step : REAL; arScrew[41].rWidth : REAL; arScrew[41].rAngle_knives : REAL; arScrew[41].rMidle_line : REAL; arScrew[41].rInstal_support : REAL; arScrew[41].rPosX0 : REAL; arScrew[41].rPosX1 : REAL; arScrew[41].rPosX2 : REAL; arScrew[41].equip.place : WSTRING(10); arScrew[41].equip.name : WSTRING(20); arScrew[41].name : WSTRING(20); arScrew[42].rRstmax : REAL; arScrew[42].rRstmin : REAL; arScrew[42].iCountCycle : INT; arScrew[42].iActuatorsMove : INT; arScrew[42].iActuatorsStep : INT; arScrew[42].iActuatorsStartPos[0] : INT; arScrew[42].iActuatorsStartPos[1] : INT; arScrew[42].support[0].bPosition : BOOL; arScrew[42].support[0].arLength[0] : INT; arScrew[42].support[0].arLength[1] : INT; arScrew[42].support[0].name : WSTRING(20); arScrew[42].support[1].bPosition : BOOL; arScrew[42].support[1].arLength[0] : INT; arScrew[42].support[1].arLength[1] : INT; arScrew[42].support[1].name : WSTRING(20); arScrew[42].bDirRotate : BOOL; arScrew[42].rOut_diam : REAL; arScrew[42].rInner_diam : REAL; arScrew[42].rTurn_step : REAL; arScrew[42].rWidth : REAL; arScrew[42].rAngle_knives : REAL; arScrew[42].rMidle_line : REAL; arScrew[42].rInstal_support : REAL; arScrew[42].rPosX0 : REAL; arScrew[42].rPosX1 : REAL; arScrew[42].rPosX2 : REAL; arScrew[42].equip.place : WSTRING(10); arScrew[42].equip.name : WSTRING(20); arScrew[42].name : WSTRING(20); arScrew[43].rRstmax : REAL; arScrew[43].rRstmin : REAL; arScrew[43].iCountCycle : INT; arScrew[43].iActuatorsMove : INT; arScrew[43].iActuatorsStep : INT; arScrew[43].iActuatorsStartPos[0] : INT; arScrew[43].iActuatorsStartPos[1] : INT; arScrew[43].support[0].bPosition : BOOL; arScrew[43].support[0].arLength[0] : INT; arScrew[43].support[0].arLength[1] : INT; arScrew[43].support[0].name : WSTRING(20); arScrew[43].support[1].bPosition : BOOL; arScrew[43].support[1].arLength[0] : INT; arScrew[43].support[1].arLength[1] : INT; arScrew[43].support[1].name : WSTRING(20); arScrew[43].bDirRotate : BOOL; arScrew[43].rOut_diam : REAL; arScrew[43].rInner_diam : REAL; arScrew[43].rTurn_step : REAL; arScrew[43].rWidth : REAL; arScrew[43].rAngle_knives : REAL; arScrew[43].rMidle_line : REAL; arScrew[43].rInstal_support : REAL; arScrew[43].rPosX0 : REAL; arScrew[43].rPosX1 : REAL; arScrew[43].rPosX2 : REAL; arScrew[43].equip.place : WSTRING(10); arScrew[43].equip.name : WSTRING(20); arScrew[43].name : WSTRING(20); arScrew[44].rRstmax : REAL; arScrew[44].rRstmin : REAL; arScrew[44].iCountCycle : INT; arScrew[44].iActuatorsMove : INT; arScrew[44].iActuatorsStep : INT; arScrew[44].iActuatorsStartPos[0] : INT; arScrew[44].iActuatorsStartPos[1] : INT; arScrew[44].support[0].bPosition : BOOL; arScrew[44].support[0].arLength[0] : INT; arScrew[44].support[0].arLength[1] : INT; arScrew[44].support[0].name : WSTRING(20); arScrew[44].support[1].bPosition : BOOL; arScrew[44].support[1].arLength[0] : INT; arScrew[44].support[1].arLength[1] : INT; arScrew[44].support[1].name : WSTRING(20); arScrew[44].bDirRotate : BOOL; arScrew[44].rOut_diam : REAL; arScrew[44].rInner_diam : REAL; arScrew[44].rTurn_step : REAL; arScrew[44].rWidth : REAL; arScrew[44].rAngle_knives : REAL; arScrew[44].rMidle_line : REAL; arScrew[44].rInstal_support : REAL; arScrew[44].rPosX0 : REAL; arScrew[44].rPosX1 : REAL; arScrew[44].rPosX2 : REAL; arScrew[44].equip.place : WSTRING(10); arScrew[44].equip.name : WSTRING(20); arScrew[44].name : WSTRING(20); arScrew[45].rRstmax : REAL; arScrew[45].rRstmin : REAL; arScrew[45].iCountCycle : INT; arScrew[45].iActuatorsMove : INT; arScrew[45].iActuatorsStep : INT; arScrew[45].iActuatorsStartPos[0] : INT; arScrew[45].iActuatorsStartPos[1] : INT; arScrew[45].support[0].bPosition : BOOL; arScrew[45].support[0].arLength[0] : INT; arScrew[45].support[0].arLength[1] : INT; arScrew[45].support[0].name : WSTRING(20); arScrew[45].support[1].bPosition : BOOL; arScrew[45].support[1].arLength[0] : INT; arScrew[45].support[1].arLength[1] : INT; arScrew[45].support[1].name : WSTRING(20); arScrew[45].bDirRotate : BOOL; arScrew[45].rOut_diam : REAL; arScrew[45].rInner_diam : REAL; arScrew[45].rTurn_step : REAL; arScrew[45].rWidth : REAL; arScrew[45].rAngle_knives : REAL; arScrew[45].rMidle_line : REAL; arScrew[45].rInstal_support : REAL; arScrew[45].rPosX0 : REAL; arScrew[45].rPosX1 : REAL; arScrew[45].rPosX2 : REAL; arScrew[45].equip.place : WSTRING(10); arScrew[45].equip.name : WSTRING(20); arScrew[45].name : WSTRING(20); arScrew[46].rRstmax : REAL; arScrew[46].rRstmin : REAL; arScrew[46].iCountCycle : INT; arScrew[46].iActuatorsMove : INT; arScrew[46].iActuatorsStep : INT; arScrew[46].iActuatorsStartPos[0] : INT; arScrew[46].iActuatorsStartPos[1] : INT; arScrew[46].support[0].bPosition : BOOL; arScrew[46].support[0].arLength[0] : INT; arScrew[46].support[0].arLength[1] : INT; arScrew[46].support[0].name : WSTRING(20); arScrew[46].support[1].bPosition : BOOL; arScrew[46].support[1].arLength[0] : INT; arScrew[46].support[1].arLength[1] : INT; arScrew[46].support[1].name : WSTRING(20); arScrew[46].bDirRotate : BOOL; arScrew[46].rOut_diam : REAL; arScrew[46].rInner_diam : REAL; arScrew[46].rTurn_step : REAL; arScrew[46].rWidth : REAL; arScrew[46].rAngle_knives : REAL; arScrew[46].rMidle_line : REAL; arScrew[46].rInstal_support : REAL; arScrew[46].rPosX0 : REAL; arScrew[46].rPosX1 : REAL; arScrew[46].rPosX2 : REAL; arScrew[46].equip.place : WSTRING(10); arScrew[46].equip.name : WSTRING(20); arScrew[46].name : WSTRING(20); arScrew[47].rRstmax : REAL; arScrew[47].rRstmin : REAL; arScrew[47].iCountCycle : INT; arScrew[47].iActuatorsMove : INT; arScrew[47].iActuatorsStep : INT; arScrew[47].iActuatorsStartPos[0] : INT; arScrew[47].iActuatorsStartPos[1] : INT; arScrew[47].support[0].bPosition : BOOL; arScrew[47].support[0].arLength[0] : INT; arScrew[47].support[0].arLength[1] : INT; arScrew[47].support[0].name : WSTRING(20); arScrew[47].support[1].bPosition : BOOL; arScrew[47].support[1].arLength[0] : INT; arScrew[47].support[1].arLength[1] : INT; arScrew[47].support[1].name : WSTRING(20); arScrew[47].bDirRotate : BOOL; arScrew[47].rOut_diam : REAL; arScrew[47].rInner_diam : REAL; arScrew[47].rTurn_step : REAL; arScrew[47].rWidth : REAL; arScrew[47].rAngle_knives : REAL; arScrew[47].rMidle_line : REAL; arScrew[47].rInstal_support : REAL; arScrew[47].rPosX0 : REAL; arScrew[47].rPosX1 : REAL; arScrew[47].rPosX2 : REAL; arScrew[47].equip.place : WSTRING(10); arScrew[47].equip.name : WSTRING(20); arScrew[47].name : WSTRING(20); arScrew[48].rRstmax : REAL; arScrew[48].rRstmin : REAL; arScrew[48].iCountCycle : INT; arScrew[48].iActuatorsMove : INT; arScrew[48].iActuatorsStep : INT; arScrew[48].iActuatorsStartPos[0] : INT; arScrew[48].iActuatorsStartPos[1] : INT; arScrew[48].support[0].bPosition : BOOL; arScrew[48].support[0].arLength[0] : INT; arScrew[48].support[0].arLength[1] : INT; arScrew[48].support[0].name : WSTRING(20); arScrew[48].support[1].bPosition : BOOL; arScrew[48].support[1].arLength[0] : INT; arScrew[48].support[1].arLength[1] : INT; arScrew[48].support[1].name : WSTRING(20); arScrew[48].bDirRotate : BOOL; arScrew[48].rOut_diam : REAL; arScrew[48].rInner_diam : REAL; arScrew[48].rTurn_step : REAL; arScrew[48].rWidth : REAL; arScrew[48].rAngle_knives : REAL; arScrew[48].rMidle_line : REAL; arScrew[48].rInstal_support : REAL; arScrew[48].rPosX0 : REAL; arScrew[48].rPosX1 : REAL; arScrew[48].rPosX2 : REAL; arScrew[48].equip.place : WSTRING(10); arScrew[48].equip.name : WSTRING(20); arScrew[48].name : WSTRING(20); arScrew[49].rRstmax : REAL; arScrew[49].rRstmin : REAL; arScrew[49].iCountCycle : INT; arScrew[49].iActuatorsMove : INT; arScrew[49].iActuatorsStep : INT; arScrew[49].iActuatorsStartPos[0] : INT; arScrew[49].iActuatorsStartPos[1] : INT; arScrew[49].support[0].bPosition : BOOL; arScrew[49].support[0].arLength[0] : INT; arScrew[49].support[0].arLength[1] : INT; arScrew[49].support[0].name : WSTRING(20); arScrew[49].support[1].bPosition : BOOL; arScrew[49].support[1].arLength[0] : INT; arScrew[49].support[1].arLength[1] : INT; arScrew[49].support[1].name : WSTRING(20); arScrew[49].bDirRotate : BOOL; arScrew[49].rOut_diam : REAL; arScrew[49].rInner_diam : REAL; arScrew[49].rTurn_step : REAL; arScrew[49].rWidth : REAL; arScrew[49].rAngle_knives : REAL; arScrew[49].rMidle_line : REAL; arScrew[49].rInstal_support : REAL; arScrew[49].rPosX0 : REAL; arScrew[49].rPosX1 : REAL; arScrew[49].rPosX2 : REAL; arScrew[49].equip.place : WSTRING(10); arScrew[49].equip.name : WSTRING(20); arScrew[49].name : WSTRING(20); arScrew[50].rRstmax : REAL; arScrew[50].rRstmin : REAL; arScrew[50].iCountCycle : INT; arScrew[50].iActuatorsMove : INT; arScrew[50].iActuatorsStep : INT; arScrew[50].iActuatorsStartPos[0] : INT; arScrew[50].iActuatorsStartPos[1] : INT; arScrew[50].support[0].bPosition : BOOL; arScrew[50].support[0].arLength[0] : INT; arScrew[50].support[0].arLength[1] : INT; arScrew[50].support[0].name : WSTRING(20); arScrew[50].support[1].bPosition : BOOL; arScrew[50].support[1].arLength[0] : INT; arScrew[50].support[1].arLength[1] : INT; arScrew[50].support[1].name : WSTRING(20); arScrew[50].bDirRotate : BOOL; arScrew[50].rOut_diam : REAL; arScrew[50].rInner_diam : REAL; arScrew[50].rTurn_step : REAL; arScrew[50].rWidth : REAL; arScrew[50].rAngle_knives : REAL; arScrew[50].rMidle_line : REAL; arScrew[50].rInstal_support : REAL; arScrew[50].rPosX0 : REAL; arScrew[50].rPosX1 : REAL; arScrew[50].rPosX2 : REAL; arScrew[50].equip.place : WSTRING(10); arScrew[50].equip.name : WSTRING(20); arScrew[50].name : WSTRING(20); arScrew[51].rRstmax : REAL; arScrew[51].rRstmin : REAL; arScrew[51].iCountCycle : INT; arScrew[51].iActuatorsMove : INT; arScrew[51].iActuatorsStep : INT; arScrew[51].iActuatorsStartPos[0] : INT; arScrew[51].iActuatorsStartPos[1] : INT; arScrew[51].support[0].bPosition : BOOL; arScrew[51].support[0].arLength[0] : INT; arScrew[51].support[0].arLength[1] : INT; arScrew[51].support[0].name : WSTRING(20); arScrew[51].support[1].bPosition : BOOL; arScrew[51].support[1].arLength[0] : INT; arScrew[51].support[1].arLength[1] : INT; arScrew[51].support[1].name : WSTRING(20); arScrew[51].bDirRotate : BOOL; arScrew[51].rOut_diam : REAL; arScrew[51].rInner_diam : REAL; arScrew[51].rTurn_step : REAL; arScrew[51].rWidth : REAL; arScrew[51].rAngle_knives : REAL; arScrew[51].rMidle_line : REAL; arScrew[51].rInstal_support : REAL; arScrew[51].rPosX0 : REAL; arScrew[51].rPosX1 : REAL; arScrew[51].rPosX2 : REAL; arScrew[51].equip.place : WSTRING(10); arScrew[51].equip.name : WSTRING(20); arScrew[51].name : WSTRING(20); arScrew[52].rRstmax : REAL; arScrew[52].rRstmin : REAL; arScrew[52].iCountCycle : INT; arScrew[52].iActuatorsMove : INT; arScrew[52].iActuatorsStep : INT; arScrew[52].iActuatorsStartPos[0] : INT; arScrew[52].iActuatorsStartPos[1] : INT; arScrew[52].support[0].bPosition : BOOL; arScrew[52].support[0].arLength[0] : INT; arScrew[52].support[0].arLength[1] : INT; arScrew[52].support[0].name : WSTRING(20); arScrew[52].support[1].bPosition : BOOL; arScrew[52].support[1].arLength[0] : INT; arScrew[52].support[1].arLength[1] : INT; arScrew[52].support[1].name : WSTRING(20); arScrew[52].bDirRotate : BOOL; arScrew[52].rOut_diam : REAL; arScrew[52].rInner_diam : REAL; arScrew[52].rTurn_step : REAL; arScrew[52].rWidth : REAL; arScrew[52].rAngle_knives : REAL; arScrew[52].rMidle_line : REAL; arScrew[52].rInstal_support : REAL; arScrew[52].rPosX0 : REAL; arScrew[52].rPosX1 : REAL; arScrew[52].rPosX2 : REAL; arScrew[52].equip.place : WSTRING(10); arScrew[52].equip.name : WSTRING(20); arScrew[52].name : WSTRING(20); arScrew[53].rRstmax : REAL; arScrew[53].rRstmin : REAL; arScrew[53].iCountCycle : INT; arScrew[53].iActuatorsMove : INT; arScrew[53].iActuatorsStep : INT; arScrew[53].iActuatorsStartPos[0] : INT; arScrew[53].iActuatorsStartPos[1] : INT; arScrew[53].support[0].bPosition : BOOL; arScrew[53].support[0].arLength[0] : INT; arScrew[53].support[0].arLength[1] : INT; arScrew[53].support[0].name : WSTRING(20); arScrew[53].support[1].bPosition : BOOL; arScrew[53].support[1].arLength[0] : INT; arScrew[53].support[1].arLength[1] : INT; arScrew[53].support[1].name : WSTRING(20); arScrew[53].bDirRotate : BOOL; arScrew[53].rOut_diam : REAL; arScrew[53].rInner_diam : REAL; arScrew[53].rTurn_step : REAL; arScrew[53].rWidth : REAL; arScrew[53].rAngle_knives : REAL; arScrew[53].rMidle_line : REAL; arScrew[53].rInstal_support : REAL; arScrew[53].rPosX0 : REAL; arScrew[53].rPosX1 : REAL; arScrew[53].rPosX2 : REAL; arScrew[53].equip.place : WSTRING(10); arScrew[53].equip.name : WSTRING(20); arScrew[53].name : WSTRING(20); arScrew[54].rRstmax : REAL; arScrew[54].rRstmin : REAL; arScrew[54].iCountCycle : INT; arScrew[54].iActuatorsMove : INT; arScrew[54].iActuatorsStep : INT; arScrew[54].iActuatorsStartPos[0] : INT; arScrew[54].iActuatorsStartPos[1] : INT; arScrew[54].support[0].bPosition : BOOL; arScrew[54].support[0].arLength[0] : INT; arScrew[54].support[0].arLength[1] : INT; arScrew[54].support[0].name : WSTRING(20); arScrew[54].support[1].bPosition : BOOL; arScrew[54].support[1].arLength[0] : INT; arScrew[54].support[1].arLength[1] : INT; arScrew[54].support[1].name : WSTRING(20); arScrew[54].bDirRotate : BOOL; arScrew[54].rOut_diam : REAL; arScrew[54].rInner_diam : REAL; arScrew[54].rTurn_step : REAL; arScrew[54].rWidth : REAL; arScrew[54].rAngle_knives : REAL; arScrew[54].rMidle_line : REAL; arScrew[54].rInstal_support : REAL; arScrew[54].rPosX0 : REAL; arScrew[54].rPosX1 : REAL; arScrew[54].rPosX2 : REAL; arScrew[54].equip.place : WSTRING(10); arScrew[54].equip.name : WSTRING(20); arScrew[54].name : WSTRING(20); arScrew[55].rRstmax : REAL; arScrew[55].rRstmin : REAL; arScrew[55].iCountCycle : INT; arScrew[55].iActuatorsMove : INT; arScrew[55].iActuatorsStep : INT; arScrew[55].iActuatorsStartPos[0] : INT; arScrew[55].iActuatorsStartPos[1] : INT; arScrew[55].support[0].bPosition : BOOL; arScrew[55].support[0].arLength[0] : INT; arScrew[55].support[0].arLength[1] : INT; arScrew[55].support[0].name : WSTRING(20); arScrew[55].support[1].bPosition : BOOL; arScrew[55].support[1].arLength[0] : INT; arScrew[55].support[1].arLength[1] : INT; arScrew[55].support[1].name : WSTRING(20); arScrew[55].bDirRotate : BOOL; arScrew[55].rOut_diam : REAL; arScrew[55].rInner_diam : REAL; arScrew[55].rTurn_step : REAL; arScrew[55].rWidth : REAL; arScrew[55].rAngle_knives : REAL; arScrew[55].rMidle_line : REAL; arScrew[55].rInstal_support : REAL; arScrew[55].rPosX0 : REAL; arScrew[55].rPosX1 : REAL; arScrew[55].rPosX2 : REAL; arScrew[55].equip.place : WSTRING(10); arScrew[55].equip.name : WSTRING(20); arScrew[55].name : WSTRING(20); arScrew[56].rRstmax : REAL; arScrew[56].rRstmin : REAL; arScrew[56].iCountCycle : INT; arScrew[56].iActuatorsMove : INT; arScrew[56].iActuatorsStep : INT; arScrew[56].iActuatorsStartPos[0] : INT; arScrew[56].iActuatorsStartPos[1] : INT; arScrew[56].support[0].bPosition : BOOL; arScrew[56].support[0].arLength[0] : INT; arScrew[56].support[0].arLength[1] : INT; arScrew[56].support[0].name : WSTRING(20); arScrew[56].support[1].bPosition : BOOL; arScrew[56].support[1].arLength[0] : INT; arScrew[56].support[1].arLength[1] : INT; arScrew[56].support[1].name : WSTRING(20); arScrew[56].bDirRotate : BOOL; arScrew[56].rOut_diam : REAL; arScrew[56].rInner_diam : REAL; arScrew[56].rTurn_step : REAL; arScrew[56].rWidth : REAL; arScrew[56].rAngle_knives : REAL; arScrew[56].rMidle_line : REAL; arScrew[56].rInstal_support : REAL; arScrew[56].rPosX0 : REAL; arScrew[56].rPosX1 : REAL; arScrew[56].rPosX2 : REAL; arScrew[56].equip.place : WSTRING(10); arScrew[56].equip.name : WSTRING(20); arScrew[56].name : WSTRING(20); arScrew[57].rRstmax : REAL; arScrew[57].rRstmin : REAL; arScrew[57].iCountCycle : INT; arScrew[57].iActuatorsMove : INT; arScrew[57].iActuatorsStep : INT; arScrew[57].iActuatorsStartPos[0] : INT; arScrew[57].iActuatorsStartPos[1] : INT; arScrew[57].support[0].bPosition : BOOL; arScrew[57].support[0].arLength[0] : INT; arScrew[57].support[0].arLength[1] : INT; arScrew[57].support[0].name : WSTRING(20); arScrew[57].support[1].bPosition : BOOL; arScrew[57].support[1].arLength[0] : INT; arScrew[57].support[1].arLength[1] : INT; arScrew[57].support[1].name : WSTRING(20); arScrew[57].bDirRotate : BOOL; arScrew[57].rOut_diam : REAL; arScrew[57].rInner_diam : REAL; arScrew[57].rTurn_step : REAL; arScrew[57].rWidth : REAL; arScrew[57].rAngle_knives : REAL; arScrew[57].rMidle_line : REAL; arScrew[57].rInstal_support : REAL; arScrew[57].rPosX0 : REAL; arScrew[57].rPosX1 : REAL; arScrew[57].rPosX2 : REAL; arScrew[57].equip.place : WSTRING(10); arScrew[57].equip.name : WSTRING(20); arScrew[57].name : WSTRING(20); arScrew[58].rRstmax : REAL; arScrew[58].rRstmin : REAL; arScrew[58].iCountCycle : INT; arScrew[58].iActuatorsMove : INT; arScrew[58].iActuatorsStep : INT; arScrew[58].iActuatorsStartPos[0] : INT; arScrew[58].iActuatorsStartPos[1] : INT; arScrew[58].support[0].bPosition : BOOL; arScrew[58].support[0].arLength[0] : INT; arScrew[58].support[0].arLength[1] : INT; arScrew[58].support[0].name : WSTRING(20); arScrew[58].support[1].bPosition : BOOL; arScrew[58].support[1].arLength[0] : INT; arScrew[58].support[1].arLength[1] : INT; arScrew[58].support[1].name : WSTRING(20); arScrew[58].bDirRotate : BOOL; arScrew[58].rOut_diam : REAL; arScrew[58].rInner_diam : REAL; arScrew[58].rTurn_step : REAL; arScrew[58].rWidth : REAL; arScrew[58].rAngle_knives : REAL; arScrew[58].rMidle_line : REAL; arScrew[58].rInstal_support : REAL; arScrew[58].rPosX0 : REAL; arScrew[58].rPosX1 : REAL; arScrew[58].rPosX2 : REAL; arScrew[58].equip.place : WSTRING(10); arScrew[58].equip.name : WSTRING(20); arScrew[58].name : WSTRING(20); arScrew[59].rRstmax : REAL; arScrew[59].rRstmin : REAL; arScrew[59].iCountCycle : INT; arScrew[59].iActuatorsMove : INT; arScrew[59].iActuatorsStep : INT; arScrew[59].iActuatorsStartPos[0] : INT; arScrew[59].iActuatorsStartPos[1] : INT; arScrew[59].support[0].bPosition : BOOL; arScrew[59].support[0].arLength[0] : INT; arScrew[59].support[0].arLength[1] : INT; arScrew[59].support[0].name : WSTRING(20); arScrew[59].support[1].bPosition : BOOL; arScrew[59].support[1].arLength[0] : INT; arScrew[59].support[1].arLength[1] : INT; arScrew[59].support[1].name : WSTRING(20); arScrew[59].bDirRotate : BOOL; arScrew[59].rOut_diam : REAL; arScrew[59].rInner_diam : REAL; arScrew[59].rTurn_step : REAL; arScrew[59].rWidth : REAL; arScrew[59].rAngle_knives : REAL; arScrew[59].rMidle_line : REAL; arScrew[59].rInstal_support : REAL; arScrew[59].rPosX0 : REAL; arScrew[59].rPosX1 : REAL; arScrew[59].rPosX2 : REAL; arScrew[59].equip.place : WSTRING(10); arScrew[59].equip.name : WSTRING(20); arScrew[59].name : WSTRING(20); arScrew[60].rRstmax : REAL; arScrew[60].rRstmin : REAL; arScrew[60].iCountCycle : INT; arScrew[60].iActuatorsMove : INT; arScrew[60].iActuatorsStep : INT; arScrew[60].iActuatorsStartPos[0] : INT; arScrew[60].iActuatorsStartPos[1] : INT; arScrew[60].support[0].bPosition : BOOL; arScrew[60].support[0].arLength[0] : INT; arScrew[60].support[0].arLength[1] : INT; arScrew[60].support[0].name : WSTRING(20); arScrew[60].support[1].bPosition : BOOL; arScrew[60].support[1].arLength[0] : INT; arScrew[60].support[1].arLength[1] : INT; arScrew[60].support[1].name : WSTRING(20); arScrew[60].bDirRotate : BOOL; arScrew[60].rOut_diam : REAL; arScrew[60].rInner_diam : REAL; arScrew[60].rTurn_step : REAL; arScrew[60].rWidth : REAL; arScrew[60].rAngle_knives : REAL; arScrew[60].rMidle_line : REAL; arScrew[60].rInstal_support : REAL; arScrew[60].rPosX0 : REAL; arScrew[60].rPosX1 : REAL; arScrew[60].rPosX2 : REAL; arScrew[60].equip.place : WSTRING(10); arScrew[60].equip.name : WSTRING(20); arScrew[60].name : WSTRING(20); arScrew[61].rRstmax : REAL; arScrew[61].rRstmin : REAL; arScrew[61].iCountCycle : INT; arScrew[61].iActuatorsMove : INT; arScrew[61].iActuatorsStep : INT; arScrew[61].iActuatorsStartPos[0] : INT; arScrew[61].iActuatorsStartPos[1] : INT; arScrew[61].support[0].bPosition : BOOL; arScrew[61].support[0].arLength[0] : INT; arScrew[61].support[0].arLength[1] : INT; arScrew[61].support[0].name : WSTRING(20); arScrew[61].support[1].bPosition : BOOL; arScrew[61].support[1].arLength[0] : INT; arScrew[61].support[1].arLength[1] : INT; arScrew[61].support[1].name : WSTRING(20); arScrew[61].bDirRotate : BOOL; arScrew[61].rOut_diam : REAL; arScrew[61].rInner_diam : REAL; arScrew[61].rTurn_step : REAL; arScrew[61].rWidth : REAL; arScrew[61].rAngle_knives : REAL; arScrew[61].rMidle_line : REAL; arScrew[61].rInstal_support : REAL; arScrew[61].rPosX0 : REAL; arScrew[61].rPosX1 : REAL; arScrew[61].rPosX2 : REAL; arScrew[61].equip.place : WSTRING(10); arScrew[61].equip.name : WSTRING(20); arScrew[61].name : WSTRING(20); arScrew[62].rRstmax : REAL; arScrew[62].rRstmin : REAL; arScrew[62].iCountCycle : INT; arScrew[62].iActuatorsMove : INT; arScrew[62].iActuatorsStep : INT; arScrew[62].iActuatorsStartPos[0] : INT; arScrew[62].iActuatorsStartPos[1] : INT; arScrew[62].support[0].bPosition : BOOL; arScrew[62].support[0].arLength[0] : INT; arScrew[62].support[0].arLength[1] : INT; arScrew[62].support[0].name : WSTRING(20); arScrew[62].support[1].bPosition : BOOL; arScrew[62].support[1].arLength[0] : INT; arScrew[62].support[1].arLength[1] : INT; arScrew[62].support[1].name : WSTRING(20); arScrew[62].bDirRotate : BOOL; arScrew[62].rOut_diam : REAL; arScrew[62].rInner_diam : REAL; arScrew[62].rTurn_step : REAL; arScrew[62].rWidth : REAL; arScrew[62].rAngle_knives : REAL; arScrew[62].rMidle_line : REAL; arScrew[62].rInstal_support : REAL; arScrew[62].rPosX0 : REAL; arScrew[62].rPosX1 : REAL; arScrew[62].rPosX2 : REAL; arScrew[62].equip.place : WSTRING(10); arScrew[62].equip.name : WSTRING(20); arScrew[62].name : WSTRING(20); arScrew[63].rRstmax : REAL; arScrew[63].rRstmin : REAL; arScrew[63].iCountCycle : INT; arScrew[63].iActuatorsMove : INT; arScrew[63].iActuatorsStep : INT; arScrew[63].iActuatorsStartPos[0] : INT; arScrew[63].iActuatorsStartPos[1] : INT; arScrew[63].support[0].bPosition : BOOL; arScrew[63].support[0].arLength[0] : INT; arScrew[63].support[0].arLength[1] : INT; arScrew[63].support[0].name : WSTRING(20); arScrew[63].support[1].bPosition : BOOL; arScrew[63].support[1].arLength[0] : INT; arScrew[63].support[1].arLength[1] : INT; arScrew[63].support[1].name : WSTRING(20); arScrew[63].bDirRotate : BOOL; arScrew[63].rOut_diam : REAL; arScrew[63].rInner_diam : REAL; arScrew[63].rTurn_step : REAL; arScrew[63].rWidth : REAL; arScrew[63].rAngle_knives : REAL; arScrew[63].rMidle_line : REAL; arScrew[63].rInstal_support : REAL; arScrew[63].rPosX0 : REAL; arScrew[63].rPosX1 : REAL; arScrew[63].rPosX2 : REAL; arScrew[63].equip.place : WSTRING(10); arScrew[63].equip.name : WSTRING(20); arScrew[63].name : WSTRING(20); arScrew[64].rRstmax : REAL; arScrew[64].rRstmin : REAL; arScrew[64].iCountCycle : INT; arScrew[64].iActuatorsMove : INT; arScrew[64].iActuatorsStep : INT; arScrew[64].iActuatorsStartPos[0] : INT; arScrew[64].iActuatorsStartPos[1] : INT; arScrew[64].support[0].bPosition : BOOL; arScrew[64].support[0].arLength[0] : INT; arScrew[64].support[0].arLength[1] : INT; arScrew[64].support[0].name : WSTRING(20); arScrew[64].support[1].bPosition : BOOL; arScrew[64].support[1].arLength[0] : INT; arScrew[64].support[1].arLength[1] : INT; arScrew[64].support[1].name : WSTRING(20); arScrew[64].bDirRotate : BOOL; arScrew[64].rOut_diam : REAL; arScrew[64].rInner_diam : REAL; arScrew[64].rTurn_step : REAL; arScrew[64].rWidth : REAL; arScrew[64].rAngle_knives : REAL; arScrew[64].rMidle_line : REAL; arScrew[64].rInstal_support : REAL; arScrew[64].rPosX0 : REAL; arScrew[64].rPosX1 : REAL; arScrew[64].rPosX2 : REAL; arScrew[64].equip.place : WSTRING(10); arScrew[64].equip.name : WSTRING(20); arScrew[64].name : WSTRING(20); arScrew[65].rRstmax : REAL; arScrew[65].rRstmin : REAL; arScrew[65].iCountCycle : INT; arScrew[65].iActuatorsMove : INT; arScrew[65].iActuatorsStep : INT; arScrew[65].iActuatorsStartPos[0] : INT; arScrew[65].iActuatorsStartPos[1] : INT; arScrew[65].support[0].bPosition : BOOL; arScrew[65].support[0].arLength[0] : INT; arScrew[65].support[0].arLength[1] : INT; arScrew[65].support[0].name : WSTRING(20); arScrew[65].support[1].bPosition : BOOL; arScrew[65].support[1].arLength[0] : INT; arScrew[65].support[1].arLength[1] : INT; arScrew[65].support[1].name : WSTRING(20); arScrew[65].bDirRotate : BOOL; arScrew[65].rOut_diam : REAL; arScrew[65].rInner_diam : REAL; arScrew[65].rTurn_step : REAL; arScrew[65].rWidth : REAL; arScrew[65].rAngle_knives : REAL; arScrew[65].rMidle_line : REAL; arScrew[65].rInstal_support : REAL; arScrew[65].rPosX0 : REAL; arScrew[65].rPosX1 : REAL; arScrew[65].rPosX2 : REAL; arScrew[65].equip.place : WSTRING(10); arScrew[65].equip.name : WSTRING(20); arScrew[65].name : WSTRING(20); arScrew[66].rRstmax : REAL; arScrew[66].rRstmin : REAL; arScrew[66].iCountCycle : INT; arScrew[66].iActuatorsMove : INT; arScrew[66].iActuatorsStep : INT; arScrew[66].iActuatorsStartPos[0] : INT; arScrew[66].iActuatorsStartPos[1] : INT; arScrew[66].support[0].bPosition : BOOL; arScrew[66].support[0].arLength[0] : INT; arScrew[66].support[0].arLength[1] : INT; arScrew[66].support[0].name : WSTRING(20); arScrew[66].support[1].bPosition : BOOL; arScrew[66].support[1].arLength[0] : INT; arScrew[66].support[1].arLength[1] : INT; arScrew[66].support[1].name : WSTRING(20); arScrew[66].bDirRotate : BOOL; arScrew[66].rOut_diam : REAL; arScrew[66].rInner_diam : REAL; arScrew[66].rTurn_step : REAL; arScrew[66].rWidth : REAL; arScrew[66].rAngle_knives : REAL; arScrew[66].rMidle_line : REAL; arScrew[66].rInstal_support : REAL; arScrew[66].rPosX0 : REAL; arScrew[66].rPosX1 : REAL; arScrew[66].rPosX2 : REAL; arScrew[66].equip.place : WSTRING(10); arScrew[66].equip.name : WSTRING(20); arScrew[66].name : WSTRING(20); arScrew[67].rRstmax : REAL; arScrew[67].rRstmin : REAL; arScrew[67].iCountCycle : INT; arScrew[67].iActuatorsMove : INT; arScrew[67].iActuatorsStep : INT; arScrew[67].iActuatorsStartPos[0] : INT; arScrew[67].iActuatorsStartPos[1] : INT; arScrew[67].support[0].bPosition : BOOL; arScrew[67].support[0].arLength[0] : INT; arScrew[67].support[0].arLength[1] : INT; arScrew[67].support[0].name : WSTRING(20); arScrew[67].support[1].bPosition : BOOL; arScrew[67].support[1].arLength[0] : INT; arScrew[67].support[1].arLength[1] : INT; arScrew[67].support[1].name : WSTRING(20); arScrew[67].bDirRotate : BOOL; arScrew[67].rOut_diam : REAL; arScrew[67].rInner_diam : REAL; arScrew[67].rTurn_step : REAL; arScrew[67].rWidth : REAL; arScrew[67].rAngle_knives : REAL; arScrew[67].rMidle_line : REAL; arScrew[67].rInstal_support : REAL; arScrew[67].rPosX0 : REAL; arScrew[67].rPosX1 : REAL; arScrew[67].rPosX2 : REAL; arScrew[67].equip.place : WSTRING(10); arScrew[67].equip.name : WSTRING(20); arScrew[67].name : WSTRING(20); arScrew[68].rRstmax : REAL; arScrew[68].rRstmin : REAL; arScrew[68].iCountCycle : INT; arScrew[68].iActuatorsMove : INT; arScrew[68].iActuatorsStep : INT; arScrew[68].iActuatorsStartPos[0] : INT; arScrew[68].iActuatorsStartPos[1] : INT; arScrew[68].support[0].bPosition : BOOL; arScrew[68].support[0].arLength[0] : INT; arScrew[68].support[0].arLength[1] : INT; arScrew[68].support[0].name : WSTRING(20); arScrew[68].support[1].bPosition : BOOL; arScrew[68].support[1].arLength[0] : INT; arScrew[68].support[1].arLength[1] : INT; arScrew[68].support[1].name : WSTRING(20); arScrew[68].bDirRotate : BOOL; arScrew[68].rOut_diam : REAL; arScrew[68].rInner_diam : REAL; arScrew[68].rTurn_step : REAL; arScrew[68].rWidth : REAL; arScrew[68].rAngle_knives : REAL; arScrew[68].rMidle_line : REAL; arScrew[68].rInstal_support : REAL; arScrew[68].rPosX0 : REAL; arScrew[68].rPosX1 : REAL; arScrew[68].rPosX2 : REAL; arScrew[68].equip.place : WSTRING(10); arScrew[68].equip.name : WSTRING(20); arScrew[68].name : WSTRING(20); arScrew[69].rRstmax : REAL; arScrew[69].rRstmin : REAL; arScrew[69].iCountCycle : INT; arScrew[69].iActuatorsMove : INT; arScrew[69].iActuatorsStep : INT; arScrew[69].iActuatorsStartPos[0] : INT; arScrew[69].iActuatorsStartPos[1] : INT; arScrew[69].support[0].bPosition : BOOL; arScrew[69].support[0].arLength[0] : INT; arScrew[69].support[0].arLength[1] : INT; arScrew[69].support[0].name : WSTRING(20); arScrew[69].support[1].bPosition : BOOL; arScrew[69].support[1].arLength[0] : INT; arScrew[69].support[1].arLength[1] : INT; arScrew[69].support[1].name : WSTRING(20); arScrew[69].bDirRotate : BOOL; arScrew[69].rOut_diam : REAL; arScrew[69].rInner_diam : REAL; arScrew[69].rTurn_step : REAL; arScrew[69].rWidth : REAL; arScrew[69].rAngle_knives : REAL; arScrew[69].rMidle_line : REAL; arScrew[69].rInstal_support : REAL; arScrew[69].rPosX0 : REAL; arScrew[69].rPosX1 : REAL; arScrew[69].rPosX2 : REAL; arScrew[69].equip.place : WSTRING(10); arScrew[69].equip.name : WSTRING(20); arScrew[69].name : WSTRING(20); arScrew[70].rRstmax : REAL; arScrew[70].rRstmin : REAL; arScrew[70].iCountCycle : INT; arScrew[70].iActuatorsMove : INT; arScrew[70].iActuatorsStep : INT; arScrew[70].iActuatorsStartPos[0] : INT; arScrew[70].iActuatorsStartPos[1] : INT; arScrew[70].support[0].bPosition : BOOL; arScrew[70].support[0].arLength[0] : INT; arScrew[70].support[0].arLength[1] : INT; arScrew[70].support[0].name : WSTRING(20); arScrew[70].support[1].bPosition : BOOL; arScrew[70].support[1].arLength[0] : INT; arScrew[70].support[1].arLength[1] : INT; arScrew[70].support[1].name : WSTRING(20); arScrew[70].bDirRotate : BOOL; arScrew[70].rOut_diam : REAL; arScrew[70].rInner_diam : REAL; arScrew[70].rTurn_step : REAL; arScrew[70].rWidth : REAL; arScrew[70].rAngle_knives : REAL; arScrew[70].rMidle_line : REAL; arScrew[70].rInstal_support : REAL; arScrew[70].rPosX0 : REAL; arScrew[70].rPosX1 : REAL; arScrew[70].rPosX2 : REAL; arScrew[70].equip.place : WSTRING(10); arScrew[70].equip.name : WSTRING(20); arScrew[70].name : WSTRING(20); arScrew[71].rRstmax : REAL; arScrew[71].rRstmin : REAL; arScrew[71].iCountCycle : INT; arScrew[71].iActuatorsMove : INT; arScrew[71].iActuatorsStep : INT; arScrew[71].iActuatorsStartPos[0] : INT; arScrew[71].iActuatorsStartPos[1] : INT; arScrew[71].support[0].bPosition : BOOL; arScrew[71].support[0].arLength[0] : INT; arScrew[71].support[0].arLength[1] : INT; arScrew[71].support[0].name : WSTRING(20); arScrew[71].support[1].bPosition : BOOL; arScrew[71].support[1].arLength[0] : INT; arScrew[71].support[1].arLength[1] : INT; arScrew[71].support[1].name : WSTRING(20); arScrew[71].bDirRotate : BOOL; arScrew[71].rOut_diam : REAL; arScrew[71].rInner_diam : REAL; arScrew[71].rTurn_step : REAL; arScrew[71].rWidth : REAL; arScrew[71].rAngle_knives : REAL; arScrew[71].rMidle_line : REAL; arScrew[71].rInstal_support : REAL; arScrew[71].rPosX0 : REAL; arScrew[71].rPosX1 : REAL; arScrew[71].rPosX2 : REAL; arScrew[71].equip.place : WSTRING(10); arScrew[71].equip.name : WSTRING(20); arScrew[71].name : WSTRING(20); arScrew[72].rRstmax : REAL; arScrew[72].rRstmin : REAL; arScrew[72].iCountCycle : INT; arScrew[72].iActuatorsMove : INT; arScrew[72].iActuatorsStep : INT; arScrew[72].iActuatorsStartPos[0] : INT; arScrew[72].iActuatorsStartPos[1] : INT; arScrew[72].support[0].bPosition : BOOL; arScrew[72].support[0].arLength[0] : INT; arScrew[72].support[0].arLength[1] : INT; arScrew[72].support[0].name : WSTRING(20); arScrew[72].support[1].bPosition : BOOL; arScrew[72].support[1].arLength[0] : INT; arScrew[72].support[1].arLength[1] : INT; arScrew[72].support[1].name : WSTRING(20); arScrew[72].bDirRotate : BOOL; arScrew[72].rOut_diam : REAL; arScrew[72].rInner_diam : REAL; arScrew[72].rTurn_step : REAL; arScrew[72].rWidth : REAL; arScrew[72].rAngle_knives : REAL; arScrew[72].rMidle_line : REAL; arScrew[72].rInstal_support : REAL; arScrew[72].rPosX0 : REAL; arScrew[72].rPosX1 : REAL; arScrew[72].rPosX2 : REAL; arScrew[72].equip.place : WSTRING(10); arScrew[72].equip.name : WSTRING(20); arScrew[72].name : WSTRING(20); arScrew[73].rRstmax : REAL; arScrew[73].rRstmin : REAL; arScrew[73].iCountCycle : INT; arScrew[73].iActuatorsMove : INT; arScrew[73].iActuatorsStep : INT; arScrew[73].iActuatorsStartPos[0] : INT; arScrew[73].iActuatorsStartPos[1] : INT; arScrew[73].support[0].bPosition : BOOL; arScrew[73].support[0].arLength[0] : INT; arScrew[73].support[0].arLength[1] : INT; arScrew[73].support[0].name : WSTRING(20); arScrew[73].support[1].bPosition : BOOL; arScrew[73].support[1].arLength[0] : INT; arScrew[73].support[1].arLength[1] : INT; arScrew[73].support[1].name : WSTRING(20); arScrew[73].bDirRotate : BOOL; arScrew[73].rOut_diam : REAL; arScrew[73].rInner_diam : REAL; arScrew[73].rTurn_step : REAL; arScrew[73].rWidth : REAL; arScrew[73].rAngle_knives : REAL; arScrew[73].rMidle_line : REAL; arScrew[73].rInstal_support : REAL; arScrew[73].rPosX0 : REAL; arScrew[73].rPosX1 : REAL; arScrew[73].rPosX2 : REAL; arScrew[73].equip.place : WSTRING(10); arScrew[73].equip.name : WSTRING(20); arScrew[73].name : WSTRING(20); arScrew[74].rRstmax : REAL; arScrew[74].rRstmin : REAL; arScrew[74].iCountCycle : INT; arScrew[74].iActuatorsMove : INT; arScrew[74].iActuatorsStep : INT; arScrew[74].iActuatorsStartPos[0] : INT; arScrew[74].iActuatorsStartPos[1] : INT; arScrew[74].support[0].bPosition : BOOL; arScrew[74].support[0].arLength[0] : INT; arScrew[74].support[0].arLength[1] : INT; arScrew[74].support[0].name : WSTRING(20); arScrew[74].support[1].bPosition : BOOL; arScrew[74].support[1].arLength[0] : INT; arScrew[74].support[1].arLength[1] : INT; arScrew[74].support[1].name : WSTRING(20); arScrew[74].bDirRotate : BOOL; arScrew[74].rOut_diam : REAL; arScrew[74].rInner_diam : REAL; arScrew[74].rTurn_step : REAL; arScrew[74].rWidth : REAL; arScrew[74].rAngle_knives : REAL; arScrew[74].rMidle_line : REAL; arScrew[74].rInstal_support : REAL; arScrew[74].rPosX0 : REAL; arScrew[74].rPosX1 : REAL; arScrew[74].rPosX2 : REAL; arScrew[74].equip.place : WSTRING(10); arScrew[74].equip.name : WSTRING(20); arScrew[74].name : WSTRING(20); arScrew[75].rRstmax : REAL; arScrew[75].rRstmin : REAL; arScrew[75].iCountCycle : INT; arScrew[75].iActuatorsMove : INT; arScrew[75].iActuatorsStep : INT; arScrew[75].iActuatorsStartPos[0] : INT; arScrew[75].iActuatorsStartPos[1] : INT; arScrew[75].support[0].bPosition : BOOL; arScrew[75].support[0].arLength[0] : INT; arScrew[75].support[0].arLength[1] : INT; arScrew[75].support[0].name : WSTRING(20); arScrew[75].support[1].bPosition : BOOL; arScrew[75].support[1].arLength[0] : INT; arScrew[75].support[1].arLength[1] : INT; arScrew[75].support[1].name : WSTRING(20); arScrew[75].bDirRotate : BOOL; arScrew[75].rOut_diam : REAL; arScrew[75].rInner_diam : REAL; arScrew[75].rTurn_step : REAL; arScrew[75].rWidth : REAL; arScrew[75].rAngle_knives : REAL; arScrew[75].rMidle_line : REAL; arScrew[75].rInstal_support : REAL; arScrew[75].rPosX0 : REAL; arScrew[75].rPosX1 : REAL; arScrew[75].rPosX2 : REAL; arScrew[75].equip.place : WSTRING(10); arScrew[75].equip.name : WSTRING(20); arScrew[75].name : WSTRING(20); arScrew[76].rRstmax : REAL; arScrew[76].rRstmin : REAL; arScrew[76].iCountCycle : INT; arScrew[76].iActuatorsMove : INT; arScrew[76].iActuatorsStep : INT; arScrew[76].iActuatorsStartPos[0] : INT; arScrew[76].iActuatorsStartPos[1] : INT; arScrew[76].support[0].bPosition : BOOL; arScrew[76].support[0].arLength[0] : INT; arScrew[76].support[0].arLength[1] : INT; arScrew[76].support[0].name : WSTRING(20); arScrew[76].support[1].bPosition : BOOL; arScrew[76].support[1].arLength[0] : INT; arScrew[76].support[1].arLength[1] : INT; arScrew[76].support[1].name : WSTRING(20); arScrew[76].bDirRotate : BOOL; arScrew[76].rOut_diam : REAL; arScrew[76].rInner_diam : REAL; arScrew[76].rTurn_step : REAL; arScrew[76].rWidth : REAL; arScrew[76].rAngle_knives : REAL; arScrew[76].rMidle_line : REAL; arScrew[76].rInstal_support : REAL; arScrew[76].rPosX0 : REAL; arScrew[76].rPosX1 : REAL; arScrew[76].rPosX2 : REAL; arScrew[76].equip.place : WSTRING(10); arScrew[76].equip.name : WSTRING(20); arScrew[76].name : WSTRING(20); arScrew[77].rRstmax : REAL; arScrew[77].rRstmin : REAL; arScrew[77].iCountCycle : INT; arScrew[77].iActuatorsMove : INT; arScrew[77].iActuatorsStep : INT; arScrew[77].iActuatorsStartPos[0] : INT; arScrew[77].iActuatorsStartPos[1] : INT; arScrew[77].support[0].bPosition : BOOL; arScrew[77].support[0].arLength[0] : INT; arScrew[77].support[0].arLength[1] : INT; arScrew[77].support[0].name : WSTRING(20); arScrew[77].support[1].bPosition : BOOL; arScrew[77].support[1].arLength[0] : INT; arScrew[77].support[1].arLength[1] : INT; arScrew[77].support[1].name : WSTRING(20); arScrew[77].bDirRotate : BOOL; arScrew[77].rOut_diam : REAL; arScrew[77].rInner_diam : REAL; arScrew[77].rTurn_step : REAL; arScrew[77].rWidth : REAL; arScrew[77].rAngle_knives : REAL; arScrew[77].rMidle_line : REAL; arScrew[77].rInstal_support : REAL; arScrew[77].rPosX0 : REAL; arScrew[77].rPosX1 : REAL; arScrew[77].rPosX2 : REAL; arScrew[77].equip.place : WSTRING(10); arScrew[77].equip.name : WSTRING(20); arScrew[77].name : WSTRING(20); arScrew[78].rRstmax : REAL; arScrew[78].rRstmin : REAL; arScrew[78].iCountCycle : INT; arScrew[78].iActuatorsMove : INT; arScrew[78].iActuatorsStep : INT; arScrew[78].iActuatorsStartPos[0] : INT; arScrew[78].iActuatorsStartPos[1] : INT; arScrew[78].support[0].bPosition : BOOL; arScrew[78].support[0].arLength[0] : INT; arScrew[78].support[0].arLength[1] : INT; arScrew[78].support[0].name : WSTRING(20); arScrew[78].support[1].bPosition : BOOL; arScrew[78].support[1].arLength[0] : INT; arScrew[78].support[1].arLength[1] : INT; arScrew[78].support[1].name : WSTRING(20); arScrew[78].bDirRotate : BOOL; arScrew[78].rOut_diam : REAL; arScrew[78].rInner_diam : REAL; arScrew[78].rTurn_step : REAL; arScrew[78].rWidth : REAL; arScrew[78].rAngle_knives : REAL; arScrew[78].rMidle_line : REAL; arScrew[78].rInstal_support : REAL; arScrew[78].rPosX0 : REAL; arScrew[78].rPosX1 : REAL; arScrew[78].rPosX2 : REAL; arScrew[78].equip.place : WSTRING(10); arScrew[78].equip.name : WSTRING(20); arScrew[78].name : WSTRING(20); arScrew[79].rRstmax : REAL; arScrew[79].rRstmin : REAL; arScrew[79].iCountCycle : INT; arScrew[79].iActuatorsMove : INT; arScrew[79].iActuatorsStep : INT; arScrew[79].iActuatorsStartPos[0] : INT; arScrew[79].iActuatorsStartPos[1] : INT; arScrew[79].support[0].bPosition : BOOL; arScrew[79].support[0].arLength[0] : INT; arScrew[79].support[0].arLength[1] : INT; arScrew[79].support[0].name : WSTRING(20); arScrew[79].support[1].bPosition : BOOL; arScrew[79].support[1].arLength[0] : INT; arScrew[79].support[1].arLength[1] : INT; arScrew[79].support[1].name : WSTRING(20); arScrew[79].bDirRotate : BOOL; arScrew[79].rOut_diam : REAL; arScrew[79].rInner_diam : REAL; arScrew[79].rTurn_step : REAL; arScrew[79].rWidth : REAL; arScrew[79].rAngle_knives : REAL; arScrew[79].rMidle_line : REAL; arScrew[79].rInstal_support : REAL; arScrew[79].rPosX0 : REAL; arScrew[79].rPosX1 : REAL; arScrew[79].rPosX2 : REAL; arScrew[79].equip.place : WSTRING(10); arScrew[79].equip.name : WSTRING(20); arScrew[79].name : WSTRING(20); arScrew[80].rRstmax : REAL; arScrew[80].rRstmin : REAL; arScrew[80].iCountCycle : INT; arScrew[80].iActuatorsMove : INT; arScrew[80].iActuatorsStep : INT; arScrew[80].iActuatorsStartPos[0] : INT; arScrew[80].iActuatorsStartPos[1] : INT; arScrew[80].support[0].bPosition : BOOL; arScrew[80].support[0].arLength[0] : INT; arScrew[80].support[0].arLength[1] : INT; arScrew[80].support[0].name : WSTRING(20); arScrew[80].support[1].bPosition : BOOL; arScrew[80].support[1].arLength[0] : INT; arScrew[80].support[1].arLength[1] : INT; arScrew[80].support[1].name : WSTRING(20); arScrew[80].bDirRotate : BOOL; arScrew[80].rOut_diam : REAL; arScrew[80].rInner_diam : REAL; arScrew[80].rTurn_step : REAL; arScrew[80].rWidth : REAL; arScrew[80].rAngle_knives : REAL; arScrew[80].rMidle_line : REAL; arScrew[80].rInstal_support : REAL; arScrew[80].rPosX0 : REAL; arScrew[80].rPosX1 : REAL; arScrew[80].rPosX2 : REAL; arScrew[80].equip.place : WSTRING(10); arScrew[80].equip.name : WSTRING(20); arScrew[80].name : WSTRING(20); arScrew[81].rRstmax : REAL; arScrew[81].rRstmin : REAL; arScrew[81].iCountCycle : INT; arScrew[81].iActuatorsMove : INT; arScrew[81].iActuatorsStep : INT; arScrew[81].iActuatorsStartPos[0] : INT; arScrew[81].iActuatorsStartPos[1] : INT; arScrew[81].support[0].bPosition : BOOL; arScrew[81].support[0].arLength[0] : INT; arScrew[81].support[0].arLength[1] : INT; arScrew[81].support[0].name : WSTRING(20); arScrew[81].support[1].bPosition : BOOL; arScrew[81].support[1].arLength[0] : INT; arScrew[81].support[1].arLength[1] : INT; arScrew[81].support[1].name : WSTRING(20); arScrew[81].bDirRotate : BOOL; arScrew[81].rOut_diam : REAL; arScrew[81].rInner_diam : REAL; arScrew[81].rTurn_step : REAL; arScrew[81].rWidth : REAL; arScrew[81].rAngle_knives : REAL; arScrew[81].rMidle_line : REAL; arScrew[81].rInstal_support : REAL; arScrew[81].rPosX0 : REAL; arScrew[81].rPosX1 : REAL; arScrew[81].rPosX2 : REAL; arScrew[81].equip.place : WSTRING(10); arScrew[81].equip.name : WSTRING(20); arScrew[81].name : WSTRING(20); arScrew[82].rRstmax : REAL; arScrew[82].rRstmin : REAL; arScrew[82].iCountCycle : INT; arScrew[82].iActuatorsMove : INT; arScrew[82].iActuatorsStep : INT; arScrew[82].iActuatorsStartPos[0] : INT; arScrew[82].iActuatorsStartPos[1] : INT; arScrew[82].support[0].bPosition : BOOL; arScrew[82].support[0].arLength[0] : INT; arScrew[82].support[0].arLength[1] : INT; arScrew[82].support[0].name : WSTRING(20); arScrew[82].support[1].bPosition : BOOL; arScrew[82].support[1].arLength[0] : INT; arScrew[82].support[1].arLength[1] : INT; arScrew[82].support[1].name : WSTRING(20); arScrew[82].bDirRotate : BOOL; arScrew[82].rOut_diam : REAL; arScrew[82].rInner_diam : REAL; arScrew[82].rTurn_step : REAL; arScrew[82].rWidth : REAL; arScrew[82].rAngle_knives : REAL; arScrew[82].rMidle_line : REAL; arScrew[82].rInstal_support : REAL; arScrew[82].rPosX0 : REAL; arScrew[82].rPosX1 : REAL; arScrew[82].rPosX2 : REAL; arScrew[82].equip.place : WSTRING(10); arScrew[82].equip.name : WSTRING(20); arScrew[82].name : WSTRING(20); arScrew[83].rRstmax : REAL; arScrew[83].rRstmin : REAL; arScrew[83].iCountCycle : INT; arScrew[83].iActuatorsMove : INT; arScrew[83].iActuatorsStep : INT; arScrew[83].iActuatorsStartPos[0] : INT; arScrew[83].iActuatorsStartPos[1] : INT; arScrew[83].support[0].bPosition : BOOL; arScrew[83].support[0].arLength[0] : INT; arScrew[83].support[0].arLength[1] : INT; arScrew[83].support[0].name : WSTRING(20); arScrew[83].support[1].bPosition : BOOL; arScrew[83].support[1].arLength[0] : INT; arScrew[83].support[1].arLength[1] : INT; arScrew[83].support[1].name : WSTRING(20); arScrew[83].bDirRotate : BOOL; arScrew[83].rOut_diam : REAL; arScrew[83].rInner_diam : REAL; arScrew[83].rTurn_step : REAL; arScrew[83].rWidth : REAL; arScrew[83].rAngle_knives : REAL; arScrew[83].rMidle_line : REAL; arScrew[83].rInstal_support : REAL; arScrew[83].rPosX0 : REAL; arScrew[83].rPosX1 : REAL; arScrew[83].rPosX2 : REAL; arScrew[83].equip.place : WSTRING(10); arScrew[83].equip.name : WSTRING(20); arScrew[83].name : WSTRING(20); arScrew[84].rRstmax : REAL; arScrew[84].rRstmin : REAL; arScrew[84].iCountCycle : INT; arScrew[84].iActuatorsMove : INT; arScrew[84].iActuatorsStep : INT; arScrew[84].iActuatorsStartPos[0] : INT; arScrew[84].iActuatorsStartPos[1] : INT; arScrew[84].support[0].bPosition : BOOL; arScrew[84].support[0].arLength[0] : INT; arScrew[84].support[0].arLength[1] : INT; arScrew[84].support[0].name : WSTRING(20); arScrew[84].support[1].bPosition : BOOL; arScrew[84].support[1].arLength[0] : INT; arScrew[84].support[1].arLength[1] : INT; arScrew[84].support[1].name : WSTRING(20); arScrew[84].bDirRotate : BOOL; arScrew[84].rOut_diam : REAL; arScrew[84].rInner_diam : REAL; arScrew[84].rTurn_step : REAL; arScrew[84].rWidth : REAL; arScrew[84].rAngle_knives : REAL; arScrew[84].rMidle_line : REAL; arScrew[84].rInstal_support : REAL; arScrew[84].rPosX0 : REAL; arScrew[84].rPosX1 : REAL; arScrew[84].rPosX2 : REAL; arScrew[84].equip.place : WSTRING(10); arScrew[84].equip.name : WSTRING(20); arScrew[84].name : WSTRING(20); arScrew[85].rRstmax : REAL; arScrew[85].rRstmin : REAL; arScrew[85].iCountCycle : INT; arScrew[85].iActuatorsMove : INT; arScrew[85].iActuatorsStep : INT; arScrew[85].iActuatorsStartPos[0] : INT; arScrew[85].iActuatorsStartPos[1] : INT; arScrew[85].support[0].bPosition : BOOL; arScrew[85].support[0].arLength[0] : INT; arScrew[85].support[0].arLength[1] : INT; arScrew[85].support[0].name : WSTRING(20); arScrew[85].support[1].bPosition : BOOL; arScrew[85].support[1].arLength[0] : INT; arScrew[85].support[1].arLength[1] : INT; arScrew[85].support[1].name : WSTRING(20); arScrew[85].bDirRotate : BOOL; arScrew[85].rOut_diam : REAL; arScrew[85].rInner_diam : REAL; arScrew[85].rTurn_step : REAL; arScrew[85].rWidth : REAL; arScrew[85].rAngle_knives : REAL; arScrew[85].rMidle_line : REAL; arScrew[85].rInstal_support : REAL; arScrew[85].rPosX0 : REAL; arScrew[85].rPosX1 : REAL; arScrew[85].rPosX2 : REAL; arScrew[85].equip.place : WSTRING(10); arScrew[85].equip.name : WSTRING(20); arScrew[85].name : WSTRING(20); arScrew[86].rRstmax : REAL; arScrew[86].rRstmin : REAL; arScrew[86].iCountCycle : INT; arScrew[86].iActuatorsMove : INT; arScrew[86].iActuatorsStep : INT; arScrew[86].iActuatorsStartPos[0] : INT; arScrew[86].iActuatorsStartPos[1] : INT; arScrew[86].support[0].bPosition : BOOL; arScrew[86].support[0].arLength[0] : INT; arScrew[86].support[0].arLength[1] : INT; arScrew[86].support[0].name : WSTRING(20); arScrew[86].support[1].bPosition : BOOL; arScrew[86].support[1].arLength[0] : INT; arScrew[86].support[1].arLength[1] : INT; arScrew[86].support[1].name : WSTRING(20); arScrew[86].bDirRotate : BOOL; arScrew[86].rOut_diam : REAL; arScrew[86].rInner_diam : REAL; arScrew[86].rTurn_step : REAL; arScrew[86].rWidth : REAL; arScrew[86].rAngle_knives : REAL; arScrew[86].rMidle_line : REAL; arScrew[86].rInstal_support : REAL; arScrew[86].rPosX0 : REAL; arScrew[86].rPosX1 : REAL; arScrew[86].rPosX2 : REAL; arScrew[86].equip.place : WSTRING(10); arScrew[86].equip.name : WSTRING(20); arScrew[86].name : WSTRING(20); arScrew[87].rRstmax : REAL; arScrew[87].rRstmin : REAL; arScrew[87].iCountCycle : INT; arScrew[87].iActuatorsMove : INT; arScrew[87].iActuatorsStep : INT; arScrew[87].iActuatorsStartPos[0] : INT; arScrew[87].iActuatorsStartPos[1] : INT; arScrew[87].support[0].bPosition : BOOL; arScrew[87].support[0].arLength[0] : INT; arScrew[87].support[0].arLength[1] : INT; arScrew[87].support[0].name : WSTRING(20); arScrew[87].support[1].bPosition : BOOL; arScrew[87].support[1].arLength[0] : INT; arScrew[87].support[1].arLength[1] : INT; arScrew[87].support[1].name : WSTRING(20); arScrew[87].bDirRotate : BOOL; arScrew[87].rOut_diam : REAL; arScrew[87].rInner_diam : REAL; arScrew[87].rTurn_step : REAL; arScrew[87].rWidth : REAL; arScrew[87].rAngle_knives : REAL; arScrew[87].rMidle_line : REAL; arScrew[87].rInstal_support : REAL; arScrew[87].rPosX0 : REAL; arScrew[87].rPosX1 : REAL; arScrew[87].rPosX2 : REAL; arScrew[87].equip.place : WSTRING(10); arScrew[87].equip.name : WSTRING(20); arScrew[87].name : WSTRING(20); arScrew[88].rRstmax : REAL; arScrew[88].rRstmin : REAL; arScrew[88].iCountCycle : INT; arScrew[88].iActuatorsMove : INT; arScrew[88].iActuatorsStep : INT; arScrew[88].iActuatorsStartPos[0] : INT; arScrew[88].iActuatorsStartPos[1] : INT; arScrew[88].support[0].bPosition : BOOL; arScrew[88].support[0].arLength[0] : INT; arScrew[88].support[0].arLength[1] : INT; arScrew[88].support[0].name : WSTRING(20); arScrew[88].support[1].bPosition : BOOL; arScrew[88].support[1].arLength[0] : INT; arScrew[88].support[1].arLength[1] : INT; arScrew[88].support[1].name : WSTRING(20); arScrew[88].bDirRotate : BOOL; arScrew[88].rOut_diam : REAL; arScrew[88].rInner_diam : REAL; arScrew[88].rTurn_step : REAL; arScrew[88].rWidth : REAL; arScrew[88].rAngle_knives : REAL; arScrew[88].rMidle_line : REAL; arScrew[88].rInstal_support : REAL; arScrew[88].rPosX0 : REAL; arScrew[88].rPosX1 : REAL; arScrew[88].rPosX2 : REAL; arScrew[88].equip.place : WSTRING(10); arScrew[88].equip.name : WSTRING(20); arScrew[88].name : WSTRING(20); arScrew[89].rRstmax : REAL; arScrew[89].rRstmin : REAL; arScrew[89].iCountCycle : INT; arScrew[89].iActuatorsMove : INT; arScrew[89].iActuatorsStep : INT; arScrew[89].iActuatorsStartPos[0] : INT; arScrew[89].iActuatorsStartPos[1] : INT; arScrew[89].support[0].bPosition : BOOL; arScrew[89].support[0].arLength[0] : INT; arScrew[89].support[0].arLength[1] : INT; arScrew[89].support[0].name : WSTRING(20); arScrew[89].support[1].bPosition : BOOL; arScrew[89].support[1].arLength[0] : INT; arScrew[89].support[1].arLength[1] : INT; arScrew[89].support[1].name : WSTRING(20); arScrew[89].bDirRotate : BOOL; arScrew[89].rOut_diam : REAL; arScrew[89].rInner_diam : REAL; arScrew[89].rTurn_step : REAL; arScrew[89].rWidth : REAL; arScrew[89].rAngle_knives : REAL; arScrew[89].rMidle_line : REAL; arScrew[89].rInstal_support : REAL; arScrew[89].rPosX0 : REAL; arScrew[89].rPosX1 : REAL; arScrew[89].rPosX2 : REAL; arScrew[89].equip.place : WSTRING(10); arScrew[89].equip.name : WSTRING(20); arScrew[89].name : WSTRING(20); arScrew[90].rRstmax : REAL; arScrew[90].rRstmin : REAL; arScrew[90].iCountCycle : INT; arScrew[90].iActuatorsMove : INT; arScrew[90].iActuatorsStep : INT; arScrew[90].iActuatorsStartPos[0] : INT; arScrew[90].iActuatorsStartPos[1] : INT; arScrew[90].support[0].bPosition : BOOL; arScrew[90].support[0].arLength[0] : INT; arScrew[90].support[0].arLength[1] : INT; arScrew[90].support[0].name : WSTRING(20); arScrew[90].support[1].bPosition : BOOL; arScrew[90].support[1].arLength[0] : INT; arScrew[90].support[1].arLength[1] : INT; arScrew[90].support[1].name : WSTRING(20); arScrew[90].bDirRotate : BOOL; arScrew[90].rOut_diam : REAL; arScrew[90].rInner_diam : REAL; arScrew[90].rTurn_step : REAL; arScrew[90].rWidth : REAL; arScrew[90].rAngle_knives : REAL; arScrew[90].rMidle_line : REAL; arScrew[90].rInstal_support : REAL; arScrew[90].rPosX0 : REAL; arScrew[90].rPosX1 : REAL; arScrew[90].rPosX2 : REAL; arScrew[90].equip.place : WSTRING(10); arScrew[90].equip.name : WSTRING(20); arScrew[90].name : WSTRING(20); arScrew[91].rRstmax : REAL; arScrew[91].rRstmin : REAL; arScrew[91].iCountCycle : INT; arScrew[91].iActuatorsMove : INT; arScrew[91].iActuatorsStep : INT; arScrew[91].iActuatorsStartPos[0] : INT; arScrew[91].iActuatorsStartPos[1] : INT; arScrew[91].support[0].bPosition : BOOL; arScrew[91].support[0].arLength[0] : INT; arScrew[91].support[0].arLength[1] : INT; arScrew[91].support[0].name : WSTRING(20); arScrew[91].support[1].bPosition : BOOL; arScrew[91].support[1].arLength[0] : INT; arScrew[91].support[1].arLength[1] : INT; arScrew[91].support[1].name : WSTRING(20); arScrew[91].bDirRotate : BOOL; arScrew[91].rOut_diam : REAL; arScrew[91].rInner_diam : REAL; arScrew[91].rTurn_step : REAL; arScrew[91].rWidth : REAL; arScrew[91].rAngle_knives : REAL; arScrew[91].rMidle_line : REAL; arScrew[91].rInstal_support : REAL; arScrew[91].rPosX0 : REAL; arScrew[91].rPosX1 : REAL; arScrew[91].rPosX2 : REAL; arScrew[91].equip.place : WSTRING(10); arScrew[91].equip.name : WSTRING(20); arScrew[91].name : WSTRING(20); arScrew[92].rRstmax : REAL; arScrew[92].rRstmin : REAL; arScrew[92].iCountCycle : INT; arScrew[92].iActuatorsMove : INT; arScrew[92].iActuatorsStep : INT; arScrew[92].iActuatorsStartPos[0] : INT; arScrew[92].iActuatorsStartPos[1] : INT; arScrew[92].support[0].bPosition : BOOL; arScrew[92].support[0].arLength[0] : INT; arScrew[92].support[0].arLength[1] : INT; arScrew[92].support[0].name : WSTRING(20); arScrew[92].support[1].bPosition : BOOL; arScrew[92].support[1].arLength[0] : INT; arScrew[92].support[1].arLength[1] : INT; arScrew[92].support[1].name : WSTRING(20); arScrew[92].bDirRotate : BOOL; arScrew[92].rOut_diam : REAL; arScrew[92].rInner_diam : REAL; arScrew[92].rTurn_step : REAL; arScrew[92].rWidth : REAL; arScrew[92].rAngle_knives : REAL; arScrew[92].rMidle_line : REAL; arScrew[92].rInstal_support : REAL; arScrew[92].rPosX0 : REAL; arScrew[92].rPosX1 : REAL; arScrew[92].rPosX2 : REAL; arScrew[92].equip.place : WSTRING(10); arScrew[92].equip.name : WSTRING(20); arScrew[92].name : WSTRING(20); arScrew[93].rRstmax : REAL; arScrew[93].rRstmin : REAL; arScrew[93].iCountCycle : INT; arScrew[93].iActuatorsMove : INT; arScrew[93].iActuatorsStep : INT; arScrew[93].iActuatorsStartPos[0] : INT; arScrew[93].iActuatorsStartPos[1] : INT; arScrew[93].support[0].bPosition : BOOL; arScrew[93].support[0].arLength[0] : INT; arScrew[93].support[0].arLength[1] : INT; arScrew[93].support[0].name : WSTRING(20); arScrew[93].support[1].bPosition : BOOL; arScrew[93].support[1].arLength[0] : INT; arScrew[93].support[1].arLength[1] : INT; arScrew[93].support[1].name : WSTRING(20); arScrew[93].bDirRotate : BOOL; arScrew[93].rOut_diam : REAL; arScrew[93].rInner_diam : REAL; arScrew[93].rTurn_step : REAL; arScrew[93].rWidth : REAL; arScrew[93].rAngle_knives : REAL; arScrew[93].rMidle_line : REAL; arScrew[93].rInstal_support : REAL; arScrew[93].rPosX0 : REAL; arScrew[93].rPosX1 : REAL; arScrew[93].rPosX2 : REAL; arScrew[93].equip.place : WSTRING(10); arScrew[93].equip.name : WSTRING(20); arScrew[93].name : WSTRING(20); arScrew[94].rRstmax : REAL; arScrew[94].rRstmin : REAL; arScrew[94].iCountCycle : INT; arScrew[94].iActuatorsMove : INT; arScrew[94].iActuatorsStep : INT; arScrew[94].iActuatorsStartPos[0] : INT; arScrew[94].iActuatorsStartPos[1] : INT; arScrew[94].support[0].bPosition : BOOL; arScrew[94].support[0].arLength[0] : INT; arScrew[94].support[0].arLength[1] : INT; arScrew[94].support[0].name : WSTRING(20); arScrew[94].support[1].bPosition : BOOL; arScrew[94].support[1].arLength[0] : INT; arScrew[94].support[1].arLength[1] : INT; arScrew[94].support[1].name : WSTRING(20); arScrew[94].bDirRotate : BOOL; arScrew[94].rOut_diam : REAL; arScrew[94].rInner_diam : REAL; arScrew[94].rTurn_step : REAL; arScrew[94].rWidth : REAL; arScrew[94].rAngle_knives : REAL; arScrew[94].rMidle_line : REAL; arScrew[94].rInstal_support : REAL; arScrew[94].rPosX0 : REAL; arScrew[94].rPosX1 : REAL; arScrew[94].rPosX2 : REAL; arScrew[94].equip.place : WSTRING(10); arScrew[94].equip.name : WSTRING(20); arScrew[94].name : WSTRING(20); arScrew[95].rRstmax : REAL; arScrew[95].rRstmin : REAL; arScrew[95].iCountCycle : INT; arScrew[95].iActuatorsMove : INT; arScrew[95].iActuatorsStep : INT; arScrew[95].iActuatorsStartPos[0] : INT; arScrew[95].iActuatorsStartPos[1] : INT; arScrew[95].support[0].bPosition : BOOL; arScrew[95].support[0].arLength[0] : INT; arScrew[95].support[0].arLength[1] : INT; arScrew[95].support[0].name : WSTRING(20); arScrew[95].support[1].bPosition : BOOL; arScrew[95].support[1].arLength[0] : INT; arScrew[95].support[1].arLength[1] : INT; arScrew[95].support[1].name : WSTRING(20); arScrew[95].bDirRotate : BOOL; arScrew[95].rOut_diam : REAL; arScrew[95].rInner_diam : REAL; arScrew[95].rTurn_step : REAL; arScrew[95].rWidth : REAL; arScrew[95].rAngle_knives : REAL; arScrew[95].rMidle_line : REAL; arScrew[95].rInstal_support : REAL; arScrew[95].rPosX0 : REAL; arScrew[95].rPosX1 : REAL; arScrew[95].rPosX2 : REAL; arScrew[95].equip.place : WSTRING(10); arScrew[95].equip.name : WSTRING(20); arScrew[95].name : WSTRING(20); arScrew[96].rRstmax : REAL; arScrew[96].rRstmin : REAL; arScrew[96].iCountCycle : INT; arScrew[96].iActuatorsMove : INT; arScrew[96].iActuatorsStep : INT; arScrew[96].iActuatorsStartPos[0] : INT; arScrew[96].iActuatorsStartPos[1] : INT; arScrew[96].support[0].bPosition : BOOL; arScrew[96].support[0].arLength[0] : INT; arScrew[96].support[0].arLength[1] : INT; arScrew[96].support[0].name : WSTRING(20); arScrew[96].support[1].bPosition : BOOL; arScrew[96].support[1].arLength[0] : INT; arScrew[96].support[1].arLength[1] : INT; arScrew[96].support[1].name : WSTRING(20); arScrew[96].bDirRotate : BOOL; arScrew[96].rOut_diam : REAL; arScrew[96].rInner_diam : REAL; arScrew[96].rTurn_step : REAL; arScrew[96].rWidth : REAL; arScrew[96].rAngle_knives : REAL; arScrew[96].rMidle_line : REAL; arScrew[96].rInstal_support : REAL; arScrew[96].rPosX0 : REAL; arScrew[96].rPosX1 : REAL; arScrew[96].rPosX2 : REAL; arScrew[96].equip.place : WSTRING(10); arScrew[96].equip.name : WSTRING(20); arScrew[96].name : WSTRING(20); arScrew[97].rRstmax : REAL; arScrew[97].rRstmin : REAL; arScrew[97].iCountCycle : INT; arScrew[97].iActuatorsMove : INT; arScrew[97].iActuatorsStep : INT; arScrew[97].iActuatorsStartPos[0] : INT; arScrew[97].iActuatorsStartPos[1] : INT; arScrew[97].support[0].bPosition : BOOL; arScrew[97].support[0].arLength[0] : INT; arScrew[97].support[0].arLength[1] : INT; arScrew[97].support[0].name : WSTRING(20); arScrew[97].support[1].bPosition : BOOL; arScrew[97].support[1].arLength[0] : INT; arScrew[97].support[1].arLength[1] : INT; arScrew[97].support[1].name : WSTRING(20); arScrew[97].bDirRotate : BOOL; arScrew[97].rOut_diam : REAL; arScrew[97].rInner_diam : REAL; arScrew[97].rTurn_step : REAL; arScrew[97].rWidth : REAL; arScrew[97].rAngle_knives : REAL; arScrew[97].rMidle_line : REAL; arScrew[97].rInstal_support : REAL; arScrew[97].rPosX0 : REAL; arScrew[97].rPosX1 : REAL; arScrew[97].rPosX2 : REAL; arScrew[97].equip.place : WSTRING(10); arScrew[97].equip.name : WSTRING(20); arScrew[97].name : WSTRING(20); arScrew[98].rRstmax : REAL; arScrew[98].rRstmin : REAL; arScrew[98].iCountCycle : INT; arScrew[98].iActuatorsMove : INT; arScrew[98].iActuatorsStep : INT; arScrew[98].iActuatorsStartPos[0] : INT; arScrew[98].iActuatorsStartPos[1] : INT; arScrew[98].support[0].bPosition : BOOL; arScrew[98].support[0].arLength[0] : INT; arScrew[98].support[0].arLength[1] : INT; arScrew[98].support[0].name : WSTRING(20); arScrew[98].support[1].bPosition : BOOL; arScrew[98].support[1].arLength[0] : INT; arScrew[98].support[1].arLength[1] : INT; arScrew[98].support[1].name : WSTRING(20); arScrew[98].bDirRotate : BOOL; arScrew[98].rOut_diam : REAL; arScrew[98].rInner_diam : REAL; arScrew[98].rTurn_step 